(* Logix 5000 project; controller PBS_Perfusion vendor 1 type 14 code 217 rev 32.14; software revision 32.03; part 13 of 27 *)
(* tags used below, declared in another part *)
   Inp_PV : BOOL;   // Input Signal (process variable) from Sensor
   Inp_PVNotify : DINT;   // Related PV object alarm prio and ack status (enum)
   Inp_Target : BOOL;   // Target State of Input (Disagree Status if not in Target State)
   Cfg_NoSubstPV : BOOL;   // 1=Disallow selection of Substitute PV
   Cfg_Debounce : REAL;   // Minimum time Input Sts must maintain state (sec)
   Set_SimPV : BOOL;   // PV used in Simulation (Inp_Sim=1)
   Sts : BOOL;   // Discrete Input Status (incl. Debounce, Manual Override, if used)
   Sts_PV : BOOL;   // Discrete Input Status (actual, not subject to Override)
   Sts_SubstPV : BOOL;   // 1=Using Substitute PV (Input being overridden)
   Sts_InpPV : BOOL;   // 1=Using Input PV (normal)
   Sts_PVBad : BOOL;   // Input Comm Status/ Quality (0=OK, 1=Bad)
   Sts_TgtDisagreeCmp : ALIAS FOR TgtDisagreeGate.Inp;   // Input vs. Target comparicon result 1=Disagree
   Sts_TgtDisagree : ALIAS FOR TgtDisagree.Inp;   // 1=Input is not in Target state
   P_DIn : BOOL;   // Unique Parameter Name for auto - discovery
   Wrk_Status : BOOL;   // Internal Status (after Manual Override selection)
   TgtDisagree : P_Alarm;   // Target Disagree Alarm
   Wrk_FallT : TIMER;   // Timer to ensure Status LOW time on falling edge
   Wrk_RiseT : TIMER;   // Timer to ensure Status HIGH time on rising edge
   Wrk_SubstPV : BOOL;   // Internal flag: Using Substitute PV
   Wrk_Sts : DINT;   // Buffer for building Val_Sts
   TgtDisagreeGate : P_Gate;   // Target Disagree Condition Gate/Delay
   MCmd_InpPV : BOOL;   // Maintenance Command to use Input PV (normal)
   MCmd_SubstPV : BOOL;   // Maintenance Command to use Substitute PV (override input)
   MRdy_InpPV : BOOL;   // 1=Ready for MCmd_InpPV (enables HMI button)
   MRdy_SubstPV : BOOL;   // 1=Ready for MCmd_SubstPV (enables HMI button)
   MSet_SubstPV : BOOL;   // Maintenance-Entered Substitute PV
   Wrk_ErrDebounce : BOOL;   // Error in Debounce Timer configuration
   REAL : DINT;
(* P_DIn, continued *)

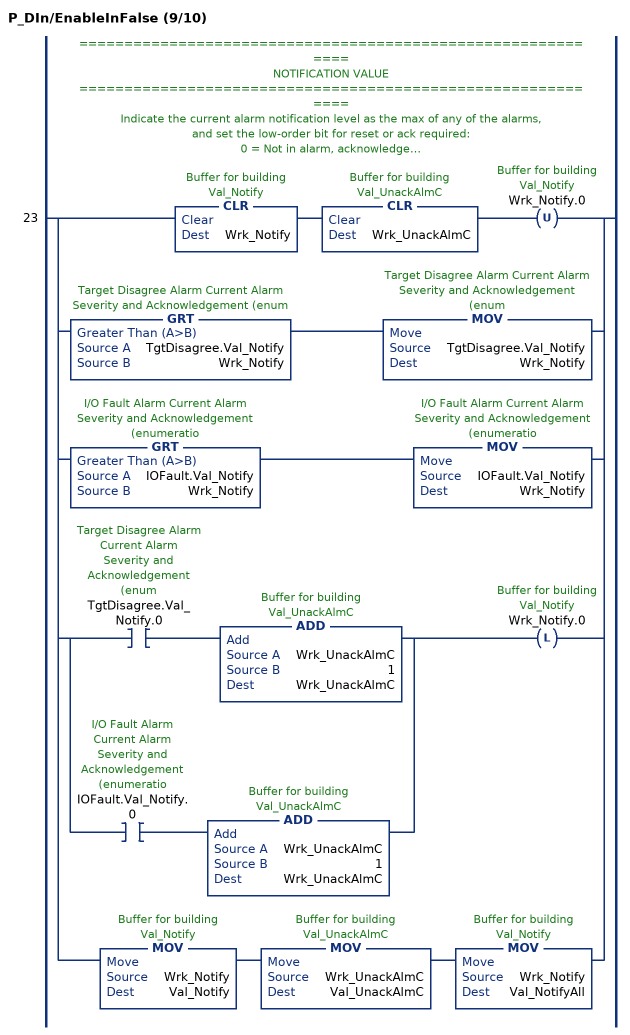
   // ============================================================
   // NOTIFICATION VALUE
   // ============================================================
   // Indicate the current alarm notification level as the max of any of the alarms,
   // and set the low-order bit for reset or ack required:
   // 0 = Not in alarm, acknowledged
   // 1 = Not in alarm, unacknowledged or reset required
   // 2 = Low severity alarm, acknowledged
   // 3 = Low severity alarm, unacknowledged
   // 4 = Medium severity alarm, acknowledged
   // 5 = Medium severity alarm, unacknowledged
   // 6 = High severity alarm, acknowledged
   // 7 = High severity alarm, unacknowledged
   // 8 = Urgent severity alarm, acknowledged
   // 9 = Urgent severity alarm, unacknowledged
   // #####  V4.00.00  2018-06-25:  Added Val_NotifyAll and Val_UnackAlmC to roll up alarm  #####
   // #####  priority / ack status and unack. alarm count.  #####
   // #####  Added I/O Fault alarm.  #####
   23: [CLR(Wrk_Notify) CLR(Wrk_UnackAlmC) OTU(Wrk_Notify.0) ,GRT(TgtDisagree.Val_Notify,Wrk_Notify) MOV(TgtDisagree.Val_Notify,Wrk_Notify) ,GRT(IOFault.Val_Notify,Wrk_Notify) MOV(IOFault.Val_Notify,Wrk_Notify) ,[XIC(TgtDisagree.Val_Notify.0) ADD(Wrk_UnackAlmC,1,Wrk_UnackAlmC) ,XIC(IOFault.Val_Notify.0) ADD(Wrk_UnackAlmC,1,Wrk_UnackAlmC) ] OTL(Wrk_Notify.0) ,MOV(Wrk_Notify,Val_Notify) MOV(Wrk_UnackAlmC,Val_UnackAlmC) MOV(Wrk_Notify,Val_NotifyAll) ];
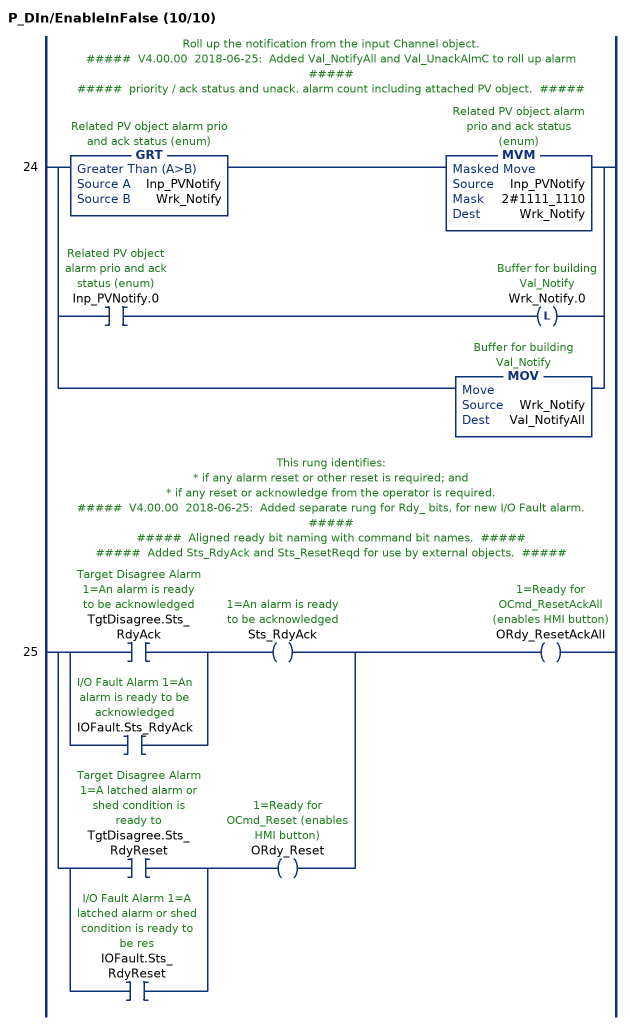
   // Roll up the notification from the input Channel object.
   // #####  V4.00.00  2018-06-25:  Added Val_NotifyAll and Val_UnackAlmC to roll up alarm  #####
   // #####  priority / ack status and unack. alarm count including attached PV object.  #####
   24: [GRT(Inp_PVNotify,Wrk_Notify) MVM(Inp_PVNotify,2#1111_1110,Wrk_Notify) ,XIC(Inp_PVNotify.0) OTL(Wrk_Notify.0) ,MOV(Wrk_Notify,Val_NotifyAll) ];
   // This rung identifies:
   // * if any alarm reset or other reset is required; and
   // * if any reset or acknowledge from the operator is required.
   // #####  V4.00.00  2018-06-25:  Added separate rung for Rdy_ bits, for new I/O Fault alarm.  #####
   // #####  Aligned ready bit naming with command bit names.  #####
   // #####  Added Sts_RdyAck and Sts_ResetReqd for use by external objects.  #####
   25: [[XIC(TgtDisagree.Sts_RdyAck) ,XIC(IOFault.Sts_RdyAck) ] OTE(Sts_RdyAck) ,[XIC(TgtDisagree.Sts_RdyReset) ,XIC(IOFault.Sts_RdyReset) ] OTE(ORdy_Reset) ]OTE(ORdy_ResetAckAll);
END_ROUTINE

ROUTINE Logic   (* ladder *)
// Normal Scan - status is updated and alarms are generated
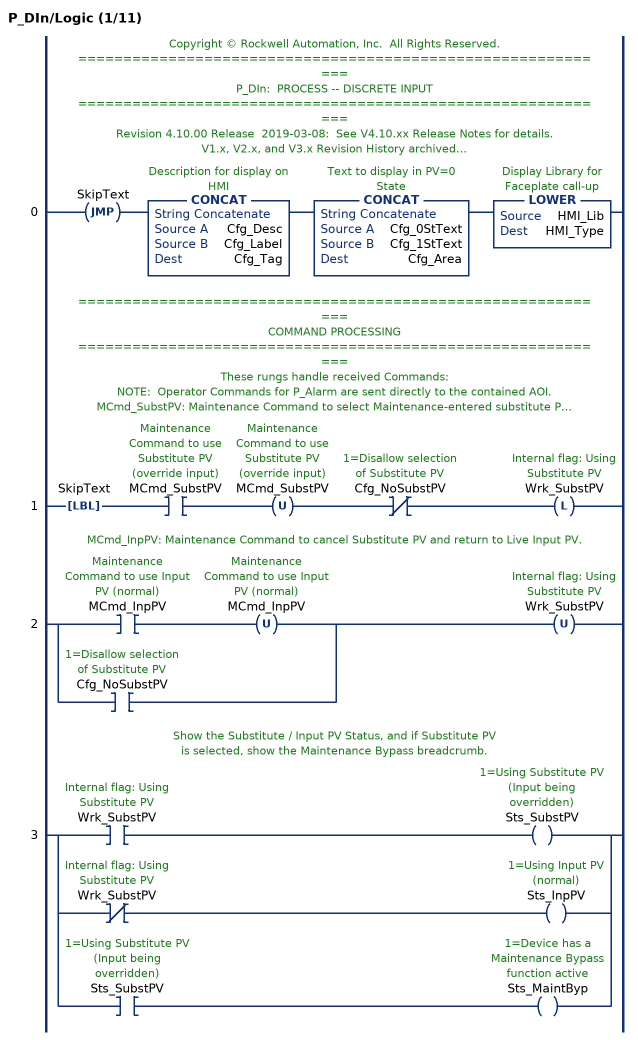
   // Copyright © Rockwell Automation, Inc.  All Rights Reserved.
   // ============================================================
   // P_DIn:  PROCESS -- DISCRETE INPUT
   // ============================================================
   // Revision 4.10.00 Release  2019-03-08:  See V4.10.xx Release Notes for details.
   // V1.x, V2.x, and V3.x Revision History archived.
   // V4.00.00  2018-06-25:  Added I/O Fault alarm.
   // Changed Inf_ items to HMI_, and added Cfg_Area for security.
   // Added notify and unack count rollup for Channel object.
   // Deleted Cfg_PCmdClear.  All Program Commands are now self-clearing.
   // Aligned ready bit naming with command bit names.
   // All OCmds/MCmds and ORdys/MRdys are now Local Tags.
   // Added Sts_RdyAck and Sts_ResetReqd for use by external objects.
   // Changed delay time configuration items to REAL seconds.
   // V4.10.00  2019-03-08:  Added Cfg_HasMoreObj.
   // ============================================================
   // This Instruction monitors a Discrete Input from a flow switch, motor vibration
   // switch, or any other discrete signal, and provides:
   // *  PV Status, with configurable names for the 0- and 1-states
   // * Input debounce for both the rising and falling transitions of the PV input
   // * An I/O Fault input.  An I/O Fault Alarm is raised when this input is true
   // *  A "Target" input -- the Target Disagree Alarm is raised when the PV input is not in
   // the same state as the Target for a configurable period of time
   // *  A Target Disagree "Gate" signal (with delay), used to enable the Alarm under
   // appropriate process conditions
   // * Commands to inhibit or enable alarms
   // * Setting of a simulated input signal for process simulation
   // * Selection of Substitute PV (by Maintenance personnel) or normal PV
   // Alarms are provided by P_Alarm AOI instances.
   // Target Disagree Status gating is provided by a P_Gate AOI instance.
   // ============================================================
   // SHOW LOCAL STRINGS
   // ============================================================
   // The STRINGs containing the text associated with each instance of this
   // instruction cannot be Input or Output Parameters, because STRINGs are not
   //  'atomic' types. (Inputs and Outputs must be SINT, INT, DINT, REAL, or BOOL.)
   // In order to make it easier to find and configure these STRINGs, this rung
   // was added.  THE JMP (and the LBL on the following rung)
   // MUST NOT BE REMOVED!!!
   // To view the STRINGs, go to the instruction instance (in LD or FBD), RIGHT-click
   // to bring up the context menu and select "Open Instruction Logic".
   // This rung will appear with the STRING values for the selected instance.
   // You may double-click the STRING values here to modify them as well.
   // #####  V4.00.00  2018-06-25:  Added string for Cfg_Area, renamed Inf_* to HMI_*.  #####
   0: JMP(SkipText)CONCAT(Cfg_Desc,Cfg_Label,Cfg_Tag)CONCAT(Cfg_0StText,Cfg_1StText,Cfg_Area)LOWER(HMI_Lib,HMI_Type);
   // ============================================================
   // COMMAND PROCESSING
   // ============================================================
   // These rungs handle received Commands:
   // NOTE:  Operator Commands for P_Alarm are sent directly to the contained AOI.
   // MCmd_SubstPV: Maintenance Command to select Maintenance-entered substitute PV
   // Do not allow this Command if Cfg_NoSubstPV is set.
   1: LBL(SkipText)XIC(MCmd_SubstPV)OTU(MCmd_SubstPV)XIO(Cfg_NoSubstPV)OTL(Wrk_SubstPV);
   // MCmd_InpPV: Maintenance Command to cancel Substitute PV and return to Live Input PV.
   2: [XIC(MCmd_InpPV) OTU(MCmd_InpPV) ,XIC(Cfg_NoSubstPV) ]OTU(Wrk_SubstPV);
   // Show the Substitute / Input PV Status, and if Substitute PV
   // is selected, show the Maintenance Bypass breadcrumb.
   3: [XIC(Wrk_SubstPV) OTE(Sts_SubstPV) ,XIO(Wrk_SubstPV) OTE(Sts_InpPV) ,XIC(Sts_SubstPV) OTE(Sts_MaintByp) ];
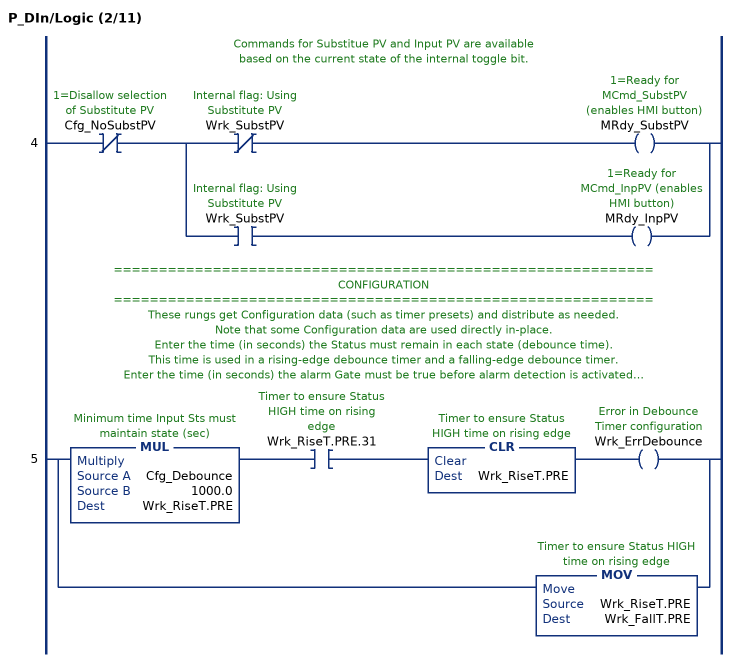
   // Commands for Substitue PV and Input PV are available
   // based on the current state of the internal toggle bit.
   4: XIO(Cfg_NoSubstPV)[XIO(Wrk_SubstPV) OTE(MRdy_SubstPV) ,XIC(Wrk_SubstPV) OTE(MRdy_InpPV) ];
   // ============================================================
   // CONFIGURATION
   // ============================================================
   // These rungs get Configuration data (such as timer presets) and distribute as needed.
   // Note that some Configuration data are used directly in-place.
   // Enter the time (in seconds) the Status must remain in each state (debounce time).
   // This time is used in a rising-edge debounce timer and a falling-edge debounce timer.
   // Enter the time (in seconds) the alarm Gate must be true before alarm detection is activated.
   // Enter the On-Delay and Off-Delay times (in seconds) for the Target Disagree Status
   // (which feeds the Target Disagree Alarm).
   // If the timer preset calcuated wraps negative (more than 2.14... million seconds), then establish
   // a valid limit value for the Preset.  Note that a negative timer preset will fault the controller!!!
   // #####  V4.00.00  2018-06-25:  Changed delay time configuration items to REAL seconds.  #####
   5: [MUL(Cfg_Debounce,1000.0,Wrk_RiseT.PRE) XIC(Wrk_RiseT.PRE.31) CLR(Wrk_RiseT.PRE) OTE(Wrk_ErrDebounce) ,MOV(Wrk_RiseT.PRE,Wrk_FallT.PRE) ];
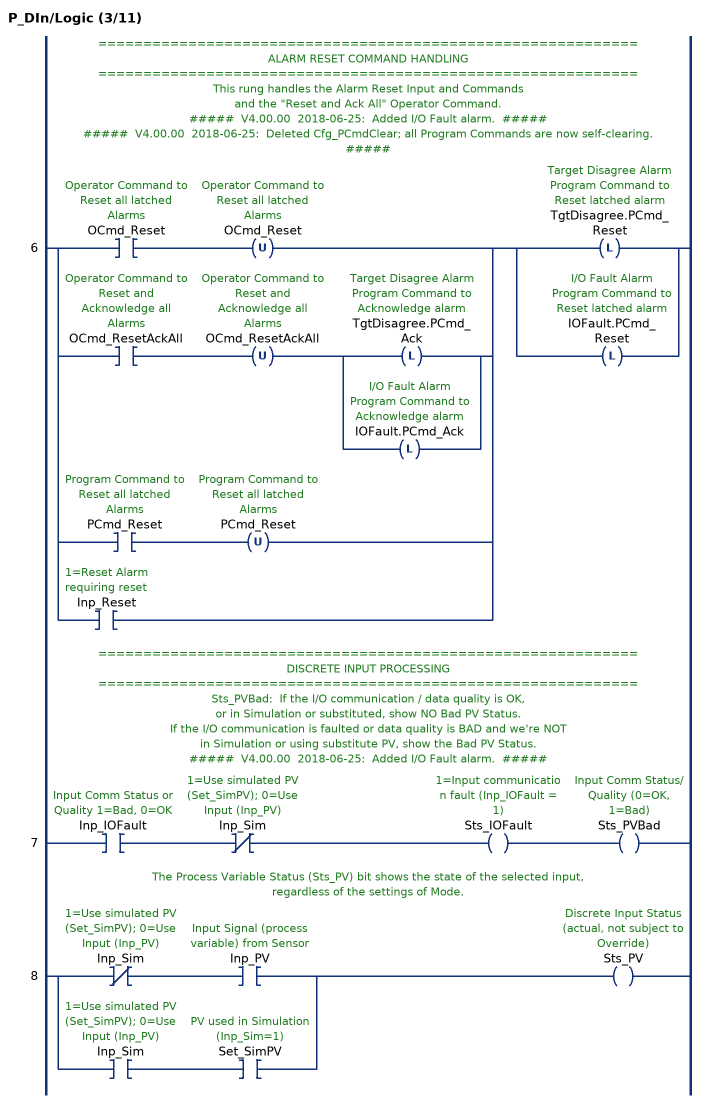
   // ============================================================
   // ALARM RESET COMMAND HANDLING
   // ============================================================
   // This rung handles the Alarm Reset Input and Commands
   // and the "Reset and Ack All" Operator Command.
   // #####  V4.00.00  2018-06-25:  Added I/O Fault alarm.  #####
   // #####  V4.00.00  2018-06-25:  Deleted Cfg_PCmdClear; all Program Commands are now self-clearing.  #####
   6: [XIC(OCmd_Reset) OTU(OCmd_Reset) ,XIC(OCmd_ResetAckAll) OTU(OCmd_ResetAckAll) [OTL(TgtDisagree.PCmd_Ack) ,OTL(IOFault.PCmd_Ack) ] ,XIC(PCmd_Reset) OTU(PCmd_Reset) ,XIC(Inp_Reset) ][OTL(TgtDisagree.PCmd_Reset) ,OTL(IOFault.PCmd_Reset) ];
   // ============================================================
   // DISCRETE INPUT PROCESSING
   // ============================================================
   // Sts_PVBad:  If the I/O communication / data quality is OK,
   // or in Simulation or substituted, show NO Bad PV Status.
   // If the I/O communication is faulted or data quality is BAD and we're NOT
   // in Simulation or using substitute PV, show the Bad PV Status.
   // #####  V4.00.00  2018-06-25:  Added I/O Fault alarm.  #####
   7: XIC(Inp_IOFault)XIO(Inp_Sim)OTE(Sts_IOFault)OTE(Sts_PVBad);
   // The Process Variable Status (Sts_PV) bit shows the state of the selected input,
   // regardless of the settings of Mode.
   8: [XIO(Inp_Sim) XIC(Inp_PV) ,XIC(Inp_Sim) XIC(Set_SimPV) ]OTE(Sts_PV);
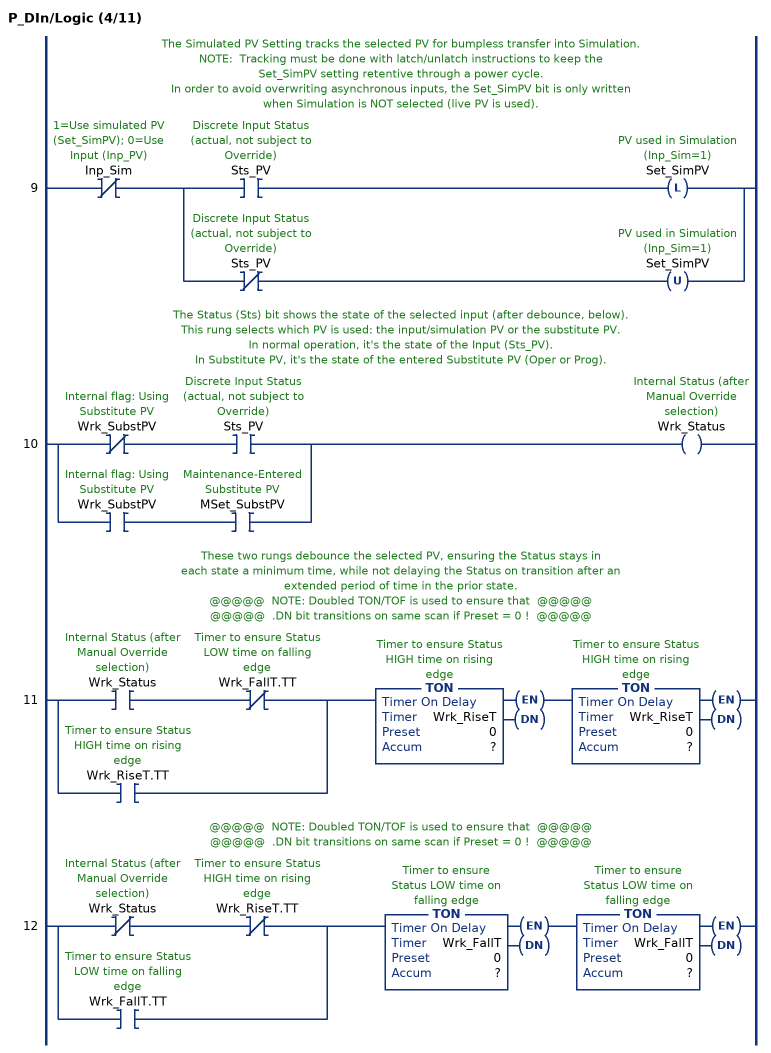
   // The Simulated PV Setting tracks the selected PV for bumpless transfer into Simulation.
   // NOTE:  Tracking must be done with latch/unlatch instructions to keep the
   // Set_SimPV setting retentive through a power cycle.
   // In order to avoid overwriting asynchronous inputs, the Set_SimPV bit is only written
   // when Simulation is NOT selected (live PV is used).
   9: XIO(Inp_Sim)[XIC(Sts_PV) OTL(Set_SimPV) ,XIO(Sts_PV) OTU(Set_SimPV) ];
   // The Status (Sts) bit shows the state of the selected input (after debounce, below).
   // This rung selects which PV is used: the input/simulation PV or the substitute PV.
   // In normal operation, it's the state of the Input (Sts_PV).
   // In Substitute PV, it's the state of the entered Substitute PV (Oper or Prog).
   10: [XIO(Wrk_SubstPV) XIC(Sts_PV) ,XIC(Wrk_SubstPV) XIC(MSet_SubstPV) ]OTE(Wrk_Status);
   // These two rungs debounce the selected PV, ensuring the Status stays in
   // each state a minimum time, while not delaying the Status on transition after an
   // extended period of time in the prior state.
   // @@@@@  NOTE: Doubled TON/TOF is used to ensure that  @@@@@
   // @@@@@  .DN bit transitions on same scan if Preset = 0 !  @@@@@
   11: [XIC(Wrk_Status) XIO(Wrk_FallT.TT) ,XIC(Wrk_RiseT.TT) ]TON(Wrk_RiseT,?,?)TON(Wrk_RiseT,?,?);
   // @@@@@  NOTE: Doubled TON/TOF is used to ensure that  @@@@@
   // @@@@@  .DN bit transitions on same scan if Preset = 0 !  @@@@@
   12: [XIO(Wrk_Status) XIO(Wrk_RiseT.TT) ,XIC(Wrk_FallT.TT) ]TON(Wrk_FallT,?,?)TON(Wrk_FallT,?,?);
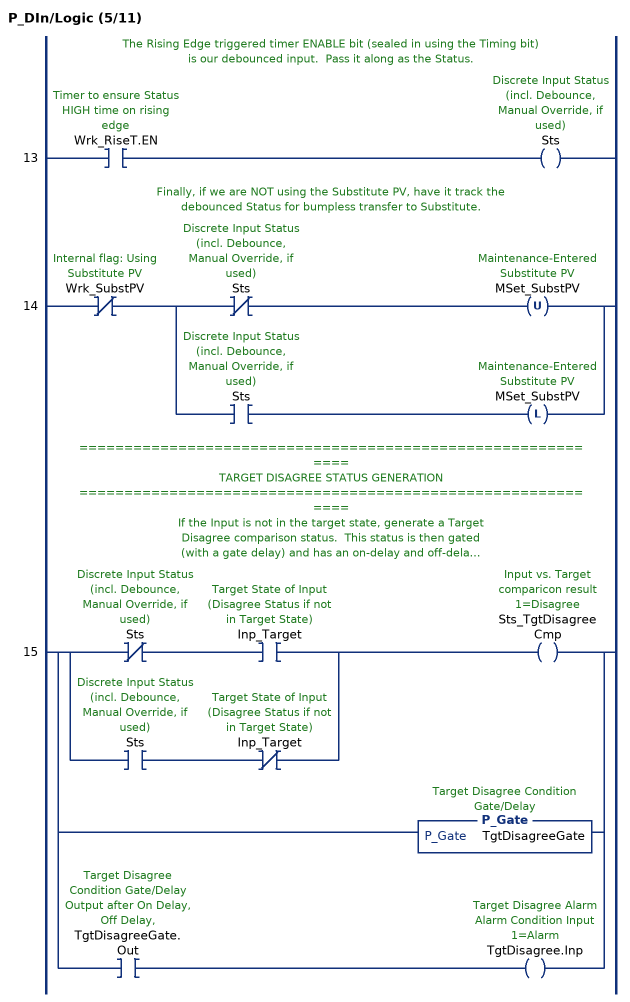
   // The Rising Edge triggered timer ENABLE bit (sealed in using the Timing bit)
   // is our debounced input.  Pass it along as the Status.
   13: XIC(Wrk_RiseT.EN)OTE(Sts);
   // Finally, if we are NOT using the Substitute PV, have it track the
   // debounced Status for bumpless transfer to Substitute.
   14: XIO(Wrk_SubstPV)[XIO(Sts) OTU(MSet_SubstPV) ,XIC(Sts) OTL(MSet_SubstPV) ];
   // ============================================================
   // TARGET DISAGREE STATUS GENERATION
   // ============================================================
   // If the Input is not in the target state, generate a Target
   // Disagree comparison status.  This status is then gated
   // (with a gate delay) and has an on-delay and off-delay
   // before feeding the final Target Disagree status bit.
   15: [[XIO(Sts) XIC(Inp_Target) ,XIC(Sts) XIO(Inp_Target) ] OTE(Sts_TgtDisagreeCmp) ,P_Gate(TgtDisagreeGate) ,XIC(TgtDisagreeGate.Out) OTE(TgtDisagree.Inp) ];
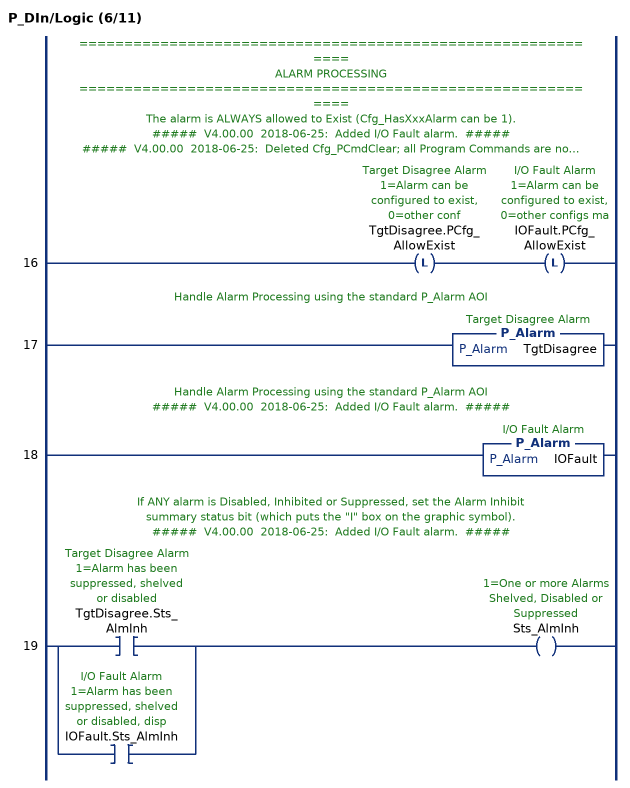
   // ============================================================
   // ALARM PROCESSING
   // ============================================================
   // The alarm is ALWAYS allowed to Exist (Cfg_HasXxxAlarm can be 1).
   // #####  V4.00.00  2018-06-25:  Added I/O Fault alarm.  #####
   // #####  V4.00.00  2018-06-25:  Deleted Cfg_PCmdClear; all Program Commands are now self-clearing.  #####
   16: OTL(TgtDisagree.PCfg_AllowExist)OTL(IOFault.PCfg_AllowExist);
   // Handle Alarm Processing using the standard P_Alarm AOI
   17: P_Alarm(TgtDisagree);
   // Handle Alarm Processing using the standard P_Alarm AOI
   // #####  V4.00.00  2018-06-25:  Added I/O Fault alarm.  #####
   18: P_Alarm(IOFault);
   // If ANY alarm is Disabled, Inhibited or Suppressed, set the Alarm Inhibit
   // summary status bit (which puts the "I" box on the graphic symbol).
   // #####  V4.00.00  2018-06-25:  Added I/O Fault alarm.  #####
   19: [XIC(TgtDisagree.Sts_AlmInh) ,XIC(IOFault.Sts_AlmInh) ]OTE(Sts_AlmInh);
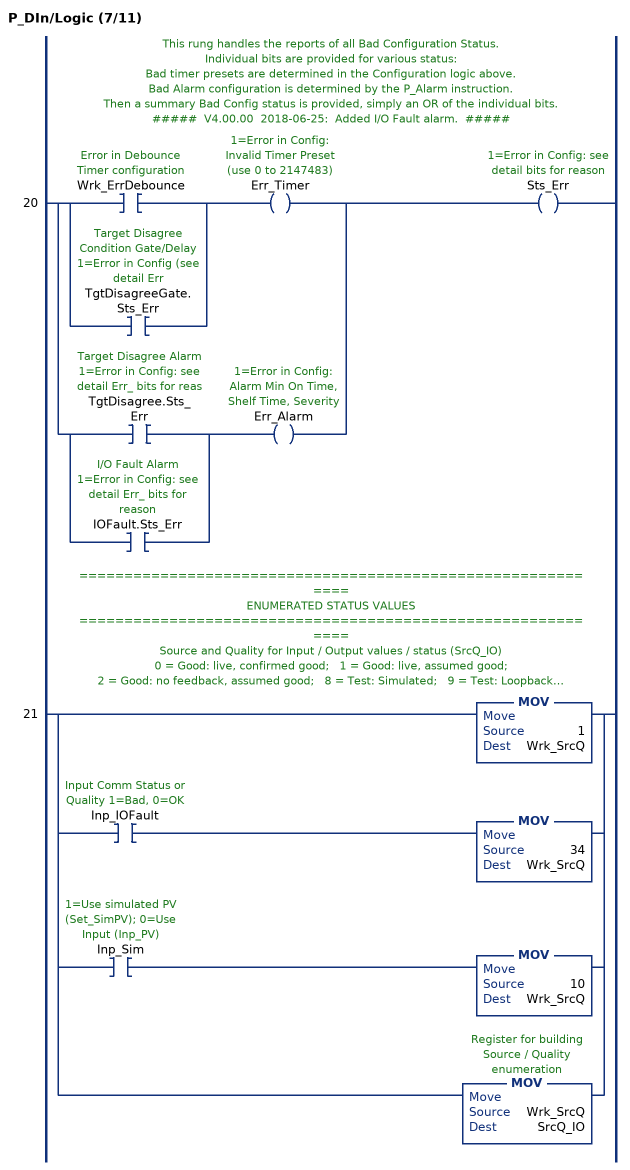
   // This rung handles the reports of all Bad Configuration Status.
   // Individual bits are provided for various status:
   // Bad timer presets are determined in the Configuration logic above.
   // Bad Alarm configuration is determined by the P_Alarm instruction.
   // Then a summary Bad Config status is provided, simply an OR of the individual bits.
   // #####  V4.00.00  2018-06-25:  Added I/O Fault alarm.  #####
   20: [[XIC(Wrk_ErrDebounce) ,XIC(TgtDisagreeGate.Sts_Err) ] OTE(Err_Timer) ,[XIC(TgtDisagree.Sts_Err) ,XIC(IOFault.Sts_Err) ] OTE(Err_Alarm) ]OTE(Sts_Err);
   // ============================================================
   // ENUMERATED STATUS VALUES
   // ============================================================
   // Source and Quality for Input / Output values / status (SrcQ_IO)
   // 0 = Good: live, confirmed good;   1 = Good: live, assumed good;
   // 2 = Good: no feedback, assumed good;   8 = Test: Simulated;   9 = Test: Loopback;
   // 10 = Test: Manually Entered;   16 = Uncertain: Live, off-spec;
   // 17 = Uncertain, Substituted at Device / Bus;   18 = Uncertain, Substituted at AOI;
   // 19 = Uncertain, using last known good;    20 = Uncertain, using replacement value;
   // 32 = Bad, Signal Failure;   33 = Bad, Channel Fault;
   // 34 = Bad, Module / Comms Fault;   35 = Bad, Invalid Configuration
   // #####  V4.00.00  2018-06-25:  Added I/O Fault alarm.  #####
   21: [MOV(1,Wrk_SrcQ) ,XIC(Inp_IOFault) MOV(34,Wrk_SrcQ) ,XIC(Inp_Sim) MOV(10,Wrk_SrcQ) ,MOV(Wrk_SrcQ,SrcQ_IO) ];
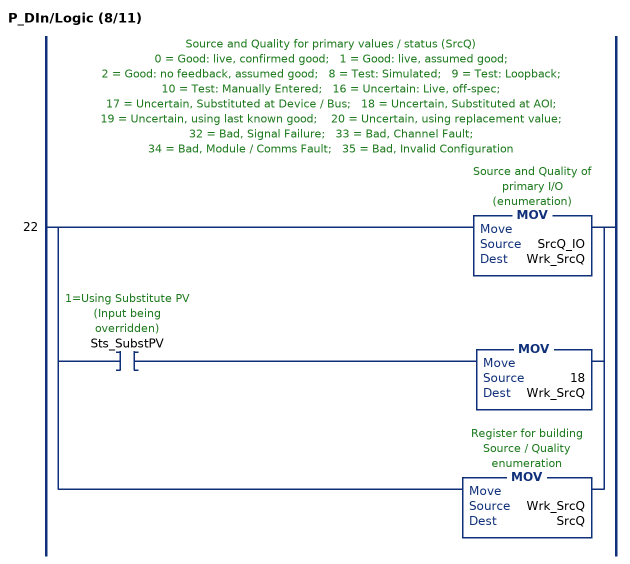
   // Source and Quality for primary values / status (SrcQ)
   // 0 = Good: live, confirmed good;   1 = Good: live, assumed good;
   // 2 = Good: no feedback, assumed good;   8 = Test: Simulated;   9 = Test: Loopback;
   // 10 = Test: Manually Entered;   16 = Uncertain: Live, off-spec;
   // 17 = Uncertain, Substituted at Device / Bus;   18 = Uncertain, Substituted at AOI;
   // 19 = Uncertain, using last known good;    20 = Uncertain, using replacement value;
   // 32 = Bad, Signal Failure;   33 = Bad, Channel Fault;
   // 34 = Bad, Module / Comms Fault;   35 = Bad, Invalid Configuration
   22: [MOV(SrcQ_IO,Wrk_SrcQ) ,XIC(Sts_SubstPV) MOV(18,Wrk_SrcQ) ,MOV(Wrk_SrcQ,SrcQ) ];
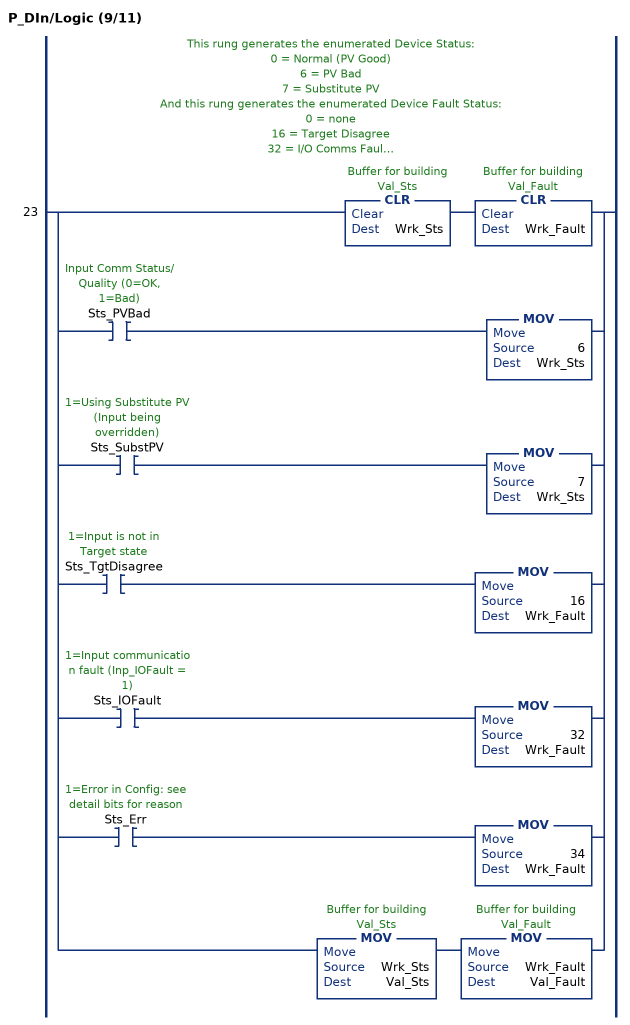
   // This rung generates the enumerated Device Status:
   // 0 = Normal (PV Good)
   // 6 = PV Bad
   // 7 = Substitute PV
   // And this rung generates the enumerated Device Fault Status:
   // 0 = none
   // 16 = Target Disagree
   // 32 = I/O Comms Fault
   // 34 = Config Error
   // #####  V4.00.00  2018-06-25:  Added I/O Fault alarm.  #####
   23: [CLR(Wrk_Sts) CLR(Wrk_Fault) ,XIC(Sts_PVBad) MOV(6,Wrk_Sts) ,XIC(Sts_SubstPV) MOV(7,Wrk_Sts) ,XIC(Sts_TgtDisagree) MOV(16,Wrk_Fault) ,XIC(Sts_IOFault) MOV(32,Wrk_Fault) ,XIC(Sts_Err) MOV(34,Wrk_Fault) ,MOV(Wrk_Sts,Val_Sts) MOV(Wrk_Fault,Val_Fault) ];
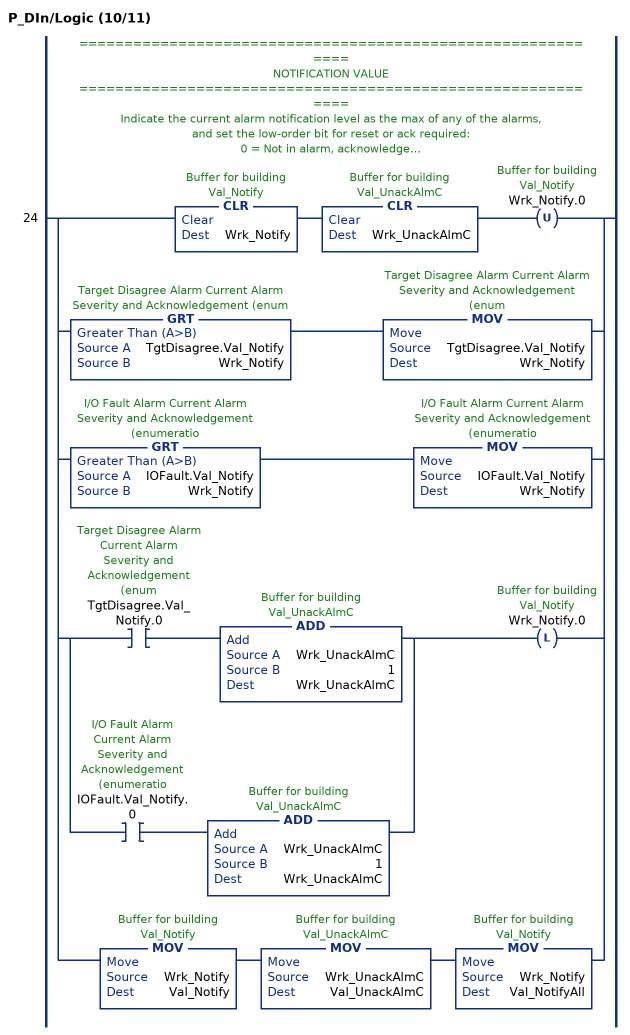
   // ============================================================
   // NOTIFICATION VALUE
   // ============================================================
   // Indicate the current alarm notification level as the max of any of the alarms,
   // and set the low-order bit for reset or ack required:
   // 0 = Not in alarm, acknowledged
   // 1 = Not in alarm, unacknowledged or reset required
   // 2 = Low severity alarm, acknowledged
   // 3 = Low severity alarm, unacknowledged
   // 4 = Medium severity alarm, acknowledged
   // 5 = Medium severity alarm, unacknowledged
   // 6 = High severity alarm, acknowledged
   // 7 = High severity alarm, unacknowledged
   // 8 = Urgent severity alarm, acknowledged
   // 9 = Urgent severity alarm, unacknowledged
   // #####  V4.00.00  2018-06-25:  Added Val_NotifyAll and Val_UnackAlmC to roll up alarm  #####
   // #####  priority / ack status and unack. alarm count.  #####
   // #####  Added I/O Fault alarm.  #####
   24: [CLR(Wrk_Notify) CLR(Wrk_UnackAlmC) OTU(Wrk_Notify.0) ,GRT(TgtDisagree.Val_Notify,Wrk_Notify) MOV(TgtDisagree.Val_Notify,Wrk_Notify) ,GRT(IOFault.Val_Notify,Wrk_Notify) MOV(IOFault.Val_Notify,Wrk_Notify) ,[XIC(TgtDisagree.Val_Notify.0) ADD(Wrk_UnackAlmC,1,Wrk_UnackAlmC) ,XIC(IOFault.Val_Notify.0) ADD(Wrk_UnackAlmC,1,Wrk_UnackAlmC) ] OTL(Wrk_Notify.0) ,MOV(Wrk_Notify,Val_Notify) MOV(Wrk_UnackAlmC,Val_UnackAlmC) MOV(Wrk_Notify,Val_NotifyAll) ];
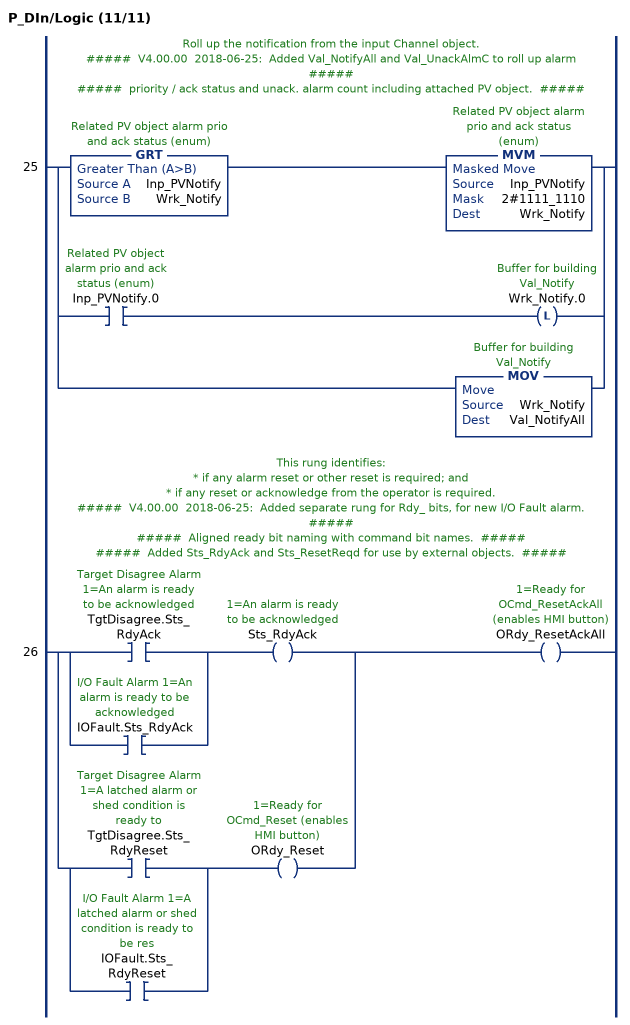
   // Roll up the notification from the input Channel object.
   // #####  V4.00.00  2018-06-25:  Added Val_NotifyAll and Val_UnackAlmC to roll up alarm  #####
   // #####  priority / ack status and unack. alarm count including attached PV object.  #####
   25: [GRT(Inp_PVNotify,Wrk_Notify) MVM(Inp_PVNotify,2#1111_1110,Wrk_Notify) ,XIC(Inp_PVNotify.0) OTL(Wrk_Notify.0) ,MOV(Wrk_Notify,Val_NotifyAll) ];
   // This rung identifies:
   // * if any alarm reset or other reset is required; and
   // * if any reset or acknowledge from the operator is required.
   // #####  V4.00.00  2018-06-25:  Added separate rung for Rdy_ bits, for new I/O Fault alarm.  #####
   // #####  Aligned ready bit naming with command bit names.  #####
   // #####  Added Sts_RdyAck and Sts_ResetReqd for use by external objects.  #####
   26: [[XIC(TgtDisagree.Sts_RdyAck) ,XIC(IOFault.Sts_RdyAck) ] OTE(Sts_RdyAck) ,[XIC(TgtDisagree.Sts_RdyReset) ,XIC(IOFault.Sts_RdyReset) ] OTE(ORdy_Reset) ]OTE(ORdy_ResetAckAll);
END_ROUTINE

ROUTINE Prescan   (* ladder *)
// Clear "lurking" Commands
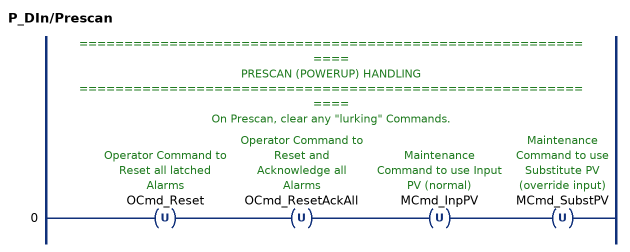
   // ============================================================
   // PRESCAN (POWERUP) HANDLING
   // ============================================================
   // On Prescan, clear any "lurking" Commands.
   0: OTU(OCmd_Reset)OTU(OCmd_ResetAckAll)OTU(MCmd_InpPV)OTU(MCmd_SubstPV);
END_ROUTINE
END_ADD_ON_INSTRUCTION

ADD_ON_INSTRUCTION P_DOut   (* revision 4.10 .01 Release, vendor Rockwell Automation, ExecutePrescan, ExecuteEnableInFalse *)
// Discrete Output
// Revision note:
// See Instruction Help for a summary of changes, and see 4.10 Release Notes for details.
// Help:
// Copyright © Rockwell Automation, Inc.  All Rights Reserved.
// This Instruction controls (and optionally monitors feedback for)
// a single Discrete Output and provides:
// *  Operator and Program Commands to:
//     -  turn the output ON
//     -  turn the output OFF
//     -  if the output is OFF, pulse it ON for a configured time
//     -  if the output is ON, pulse it OFF for a configured time, and
//     -  pulse the output continuously at the configured ON
//         and OFF times (e.g., for blinking a lamp)
// *  User-configurable ON delay and OFF delay before first output change
// *  User-configurable text labels for the ON and OFF states
// *  Optional monitoring of ON and OFF state confirmation feedbacks
// *  Detection of Failure to turn ON or OFF (when feedbacks are used)
// *  Monitoring of Permissive conditions to allow energizing output
// *  Monitoring of Interlock conditions to de-energize output
// *  Simulation, providing feedback of a working device while
//       disabling output (keeping de-energized)
// *  Monitoring of I/O communication faults
// *  Alarms for Fail to Turn ON, Fail to turn OFF (if feedbacks are
//       used), Interlock Trip, I/O Fault
// *  "NotReady" status for display on Graphic Symbol and "Available"
//      status for use by automation logic to know whether output can be
//      controlled by other objects.
// Command Sources are arbitrated by a P_CmdSrc Add-On Instruction instance.
// Command Sources: Operator, Program, External, Override, Maintenance, Out of
// Service, Hand.  Alarms are provided by P_Alarm Add-On Instruction instances.
// SUMMARY OF CHANGES FROM PREVIOUS VERSION (4.10.00)
// * Corrected operation of state machine with alert horn.
// SUMMARY OF CHANGES FROM PREVIOUS VERSION (4.00.02)
// See 4.10 Release Notes for details.
// * Added audible alert on commanded energize/state change.
// * Added Horn Status, Horn Inhibit.
// * Changed availability to use input availability from interlocks.
// * Updated to P_CmdSrc V4.10.00.
// * Added Cfg_HasMoreObj.
// SUMMARY OF CHANGES FROM PREVIOUS VERSION (4.00.00)
// See 4.00 Release Notes for details.
// * Fixed feedback determination for simulation or no feedback.
// SUMMARY OF CHANGES FROM PREVIOUS VERSION (3.5-11)
// See 4.00 Release Notes for details.
// * Changed Inf_ items to HMI_, and added Cfg_Area for security.
// * Added notify and unack count rollup for associated object(s).
// * Changed "Mode" to "Command Source" using P_CmdSrc 4.00.00.
// * Deleted Cfg_PCmdClear; all Program Commands are now self-clearing.
// * Added option Cfg_HasPulse to enable or disable pulsing functions.
// * Aligned ready bit naming with command bit names.
// * All OCmds/MCmds and ORdys/MRdys are now Local Tags.
// * Added Sts_RdyAck and Sts_RdyReset for use by external objects.
// * Changed delay / time configuration items to REAL seconds.
VAR_INPUT
   Inp_OnFdbk : BOOL; {visible}   // Input Signal: ON feedback from device
   Inp_OffFdbk : BOOL; {visible}   // Input Signal: OFF feedback from device
   Inp_PermOK : BOOL := 1; {visible}   // 1=ON Permissives OK, device can turn ON
   Inp_NBPermOK : BOOL := 1; {visible}   // 1=Non-Bypassable ON Permissives OK, device can turn ON
   Inp_IntlkOK : BOOL := 1; {visible}   // 1=Interlocks OK, device can turn ON and stay ON
   Inp_NBIntlkOK : BOOL := 1; {visible}   // 1=Non-Bypassable Interlocks OK, device can turn ON and stay ON
   Inp_IntlkAvail : BOOL;   // 1 = Interlock Availibility OK
   Inp_IOFault : BOOL;   // Input Communication Status 0=OK, 1=fail
   Inp_Sim : BOOL;   // 1=Simulate working device; 0=Turn ON/OFF actual device
   Inp_Hand : ALIAS FOR CmdSrc.Inp_Hand;
   Inp_Ovrd : ALIAS FOR CmdSrc.Inp_Ovrd;
   Inp_OvrdCmd : DINT;   // Ovrd Device Command 0=None, 1=Off, 2=On, 3=Pulse Off, 4=Pulse On, 5=Pulse Cont
   Inp_ExtInh : ALIAS FOR CmdSrc.Inp_ExtInh;
   Inp_HornInh : BOOL;   // 1 = Inhibit audible alert, 0 = Alllow audible alert
   Inp_Reset : BOOL;   // 1=Reset Shed Latches and Cleared Alarms
   Cfg_HasPulse : BOOL;   // 1=Enable pulsing functions, 0=On/Off only
   Cfg_CompletePulse : BOOL;   // 1=Finish Pulse when commanded ON or OFF; 0=switch immediately
   Cfg_HasOnFdbk : BOOL;   // 1=Device provides an ON feedback signal
   Cfg_HasOffFdbk : BOOL;   // 1=Device provides an OFF feedback signal
   Cfg_UseOnFdbk : BOOL;   // 1=Device ON feedback should be used for failure checking
   Cfg_UseOffFdbk : BOOL;   // 1=Device OFF feedback should be used for failure checking
   Cfg_FdbkFail : BOOL;   // 1=Both feedbacks ON is invalid; 0=Both feedbacks OFF is invalid
   Cfg_HasPermObj : BOOL;   // 1=Tells HMI a P_Perm is connected to Inp_Perm
   Cfg_HasIntlkObj : BOOL;   // 1=Tells HMI a P_Intlk is connected to Inp_Intlk
   Cfg_HasMoreObj : BOOL;   // 1=Tells HMI an object with more info is available
   Cfg_HornOnChange : BOOL;   // 0 = Horn on energize only, 1 = Horn on any state change
   Cfg_OperOffPrio : BOOL;   // 1=OCmd_Off any time, 0=OCmd_Off only when Oper selected
   Cfg_ExtOffPrio : BOOL;   // 1=XCmd_Off any time, 0=XCmd_Off only when Oper selected
   Cfg_OCmdResets : BOOL;   // 1=New device OCmd resets shed latches and cleared alarms, 0=OCmdReset req'd.
   Cfg_XCmdResets : BOOL;   // 1=New device XCmd resets shed latches and cleared alarms, 0=XCmdReset req'd.
   Cfg_OvrdPermIntlk : BOOL;   // 1=Override ignores Bypassable Perm/ Intlk; 0=always use Perm/Intlk
   Cfg_ShedOnFail : BOOL := 1;   // 1=Go to State 0 and Alarm on Fail to reach position; 0=Alarm only on Fail
   Cfg_ShedOnIOFault : BOOL := 1;   // 1=Go to State 0 and Alarm on I/O Fault; 0=Alarm only on I/O Fault
   Cfg_HasOnFailAlm : ALIAS FOR OnFail.Cfg_Exists;   // 1=Fail to Turn ON Alarm exists and will be checked
   Cfg_HasOffFailAlm : ALIAS FOR OffFail.Cfg_Exists;   // 1=Fail to Turn OFF Alarm exists and will be checked
   Cfg_HasIntlkTripAlm : ALIAS FOR IntlkTrip.Cfg_Exists;   // 1=Interlock Trip Alarm exists and will be checked
   Cfg_HasIOFaultAlm : ALIAS FOR IOFault.Cfg_Exists;   // 1=I/O Fault Alarm exists and will be checked
   Cfg_OnFailResetReqd : ALIAS FOR OnFail.Cfg_ResetReqd;   // 1=Reset required to clear Fail to Turn ON Alarm
   Cfg_OffFailResetReqd : ALIAS FOR OffFail.Cfg_ResetReqd;   // 1=Reset required to clear Fail to Turn OFF Alarm
   Cfg_IntlkTripResetReqd : ALIAS FOR IntlkTrip.Cfg_ResetReqd;   // 1=Reset required to clear Interlock Trip Alarm
   Cfg_IOFaultResetReqd : ALIAS FOR IOFault.Cfg_ResetReqd;   // 1=Reset required to clear I/O Fault Alarm
   Cfg_OnFailAckReqd : ALIAS FOR OnFail.Cfg_AckReqd;   // 1=Acknowledge required for Fail to Turn ON Alarm
   Cfg_OffFailAckReqd : ALIAS FOR OffFail.Cfg_AckReqd;   // 1=Acknowledge required for Fail to Turn OFF Alarm
   Cfg_IntlkTripAckReqd : ALIAS FOR IntlkTrip.Cfg_AckReqd;   // 1=Acknowledge required for Interlock Trip Alarm
   Cfg_IOFaultAckReqd : ALIAS FOR IOFault.Cfg_AckReqd;   // 1=Acknowledge required for I/O Fault Alarm
   Cfg_OnFailSeverity : ALIAS FOR OnFail.Cfg_Severity;   // Fail To Turn OFF Alarm Severity: 1..250=Low, 251..500=Medium, 501..750=High, 751..1000=Urgent
   Cfg_OffFailSeverity : ALIAS FOR OffFail.Cfg_Severity;   // Fail To Turn ON Alarm Severity: 1..250=Low, 251..500=Medium, 501..750=High, 751..1000=Urgent
   Cfg_IntlkTripSeverity : ALIAS FOR IntlkTrip.Cfg_Severity;   // Interlock Trip Alarm Severity: 1..250=Low, 251..500=Medium, 501..750=High, 751..1000=Urgent
   Cfg_IOFaultSeverity : ALIAS FOR IOFault.Cfg_Severity;   // I/O Fault Alarm Severity: 1..250=Low, 251..500=Medium, 501..750=High, 751..1000=Urgent
   Cfg_StartHornT : REAL;   // Time to sound audible on commanded start (sec) (0=disabled)
   Cfg_SimFdbkT : REAL := 2.0;   // Delay to echo back of ON/OFF status when in Simulation (sec)
   Cfg_OnDelayT : REAL;   // Delay before initially turning output ON (sec)
   Cfg_OffDelayT : REAL;   // Delay before initially turning output OFF (sec)
   Cfg_OnPulseT : REAL := 0.5;   // Output ON time for Pulse ON or Pulse Continuous
   Cfg_OffPulseT : REAL := 0.5;   // Output OFF time for Pulse OFF or Pulse Continuous
   Cfg_OnFailT : REAL := 10.0;   // Time after Output ON to get ON Feedback before Fault (sec)
   Cfg_OffFailT : REAL := 10.0;   // Time after Output OFF to get OFF Feedback before Fault (sec)
   PSet_Owner : DINT;   // Program Owner Request ID (non-zero) or Release (zero)
   PCmd_On : BOOL;   // Program Command to turn device ON
   PCmd_Off : BOOL;   // Program Command to turn device OFF
   PCmd_OnPulse : BOOL;   // Program Command to pulse device (which is OFF) ON once
   PCmd_OffPulse : BOOL;   // Program Command to pulse device (which is ON) OFF once
   PCmd_ContPulse : BOOL;   // Program Command to pulse device continuously (blink)
   PCmd_Prog : ALIAS FOR CmdSrc.PCmd_Prog;
   PCmd_Oper : ALIAS FOR CmdSrc.PCmd_Oper;
   PCmd_Lock : ALIAS FOR CmdSrc.PCmd_Lock;
   PCmd_Unlock : ALIAS FOR CmdSrc.PCmd_Unlock;
   PCmd_Normal : ALIAS FOR CmdSrc.PCmd_Normal;
   PCmd_Reset : BOOL;   // Program Command to ResetShed Latches and Cleared Alarms
   PCmd_OnFailAck : ALIAS FOR OnFail.PCmd_Ack;   // Program Command to Acknowledge Fail to Turn ON Alarm
   PCmd_OnFailSuppress : ALIAS FOR OnFail.PCmd_Suppress;   // Program Command to Suppress Fail to Turn ON Alarm
   PCmd_OnFailUnsuppress : ALIAS FOR OnFail.PCmd_Unsuppress;   // Program Command to UnsuppressFail to Turn ON Alarm
   PCmd_OnFailUnshelve : ALIAS FOR OnFail.PCmd_Unshelve;   // Program Command to Unshelve Fail to Turn ON Alarm
   PCmd_OffFailAck : ALIAS FOR OffFail.PCmd_Ack;   // Program Command to Acknowledge Fail to Turn OFF Alarm
   PCmd_OffFailSuppress : ALIAS FOR OffFail.PCmd_Suppress;   // Program Command to Suppress Fail to Turn OFF Alarm
   PCmd_OffFailUnsuppress : ALIAS FOR OffFail.PCmd_Unsuppress;   // Program Command to Unsuppress Fail to Turn OFF Alarm
   PCmd_OffFailUnshelve : ALIAS FOR OffFail.PCmd_Unshelve;   // Program Command to Unshelve Failt to Turn OFF Alarm
   PCmd_IntlkTripAck : ALIAS FOR IntlkTrip.PCmd_Ack;   // Program Command to Acknowledge Interlock Trip Alarm
   PCmd_IntlkTripSuppress : ALIAS FOR IntlkTrip.PCmd_Suppress;   // Program Command to Suppress Interlock Trip Alarm
   PCmd_IntlkTripUnsuppress : ALIAS FOR IntlkTrip.PCmd_Unsuppress;   // Program Command to Unsuppress Interlock Trip Alarm
   PCmd_IntlkTripUnshelve : ALIAS FOR IntlkTrip.PCmd_Unshelve;   // Program Command to Unshelve Interlock Trip Alarm
   PCmd_IOFaultAck : ALIAS FOR IOFault.PCmd_Ack;   // Program Command to Acknowledge I/O Fault Alarm
   PCmd_IOFaultSuppress : ALIAS FOR IOFault.PCmd_Suppress;   // Program Command to Suppress I/O Fault Alarm
   PCmd_IOFaultUnsuppress : ALIAS FOR IOFault.PCmd_Unsuppress;   // Program Command to Unsuppress I/O Fault Alarm
   PCmd_IOFaultUnshelve : ALIAS FOR IOFault.PCmd_Unshelve;   // Program Command to Unshelve I/O Fault Alarm
   MCmd_Rel : ALIAS FOR CmdSrc.MCmd_Rel;
   OCmd_Unlock : ALIAS FOR CmdSrc.OCmd_Unlock;
   XCmd_On : BOOL;   // External Command to turn device ON
   XCmd_Off : BOOL;   // External Command to turn device OFF
   XCmd_OnPulse : BOOL;   // External Command to pulse device (which is OFF) ON once
   XCmd_OffPulse : BOOL;   // External Command to pulse device (which is ON) OFF once
   XCmd_ContPulse : BOOL;   // External Command to pulse device continuously (blink)
   XCmd_Acq : ALIAS FOR CmdSrc.XCmd_Acq;
   XCmd_Rel : ALIAS FOR CmdSrc.XCmd_Rel;
   XCmd_Reset : BOOL;   // Ext Cmd to clear shed latches and cleared alarms
END_VAR
VAR_OUTPUT
   Out : BOOL; {access Read Only, visible}   // Primary Output 1=ON, 0=OFF
   Out_Horn : BOOL; {access Read Only, visible}   // 1=Sound audible prior to commanded energize/ state change
   SrcQ_IO : DINT; {access Read Only}   // Source and Quality of primary I/O (enumeration)
   SrcQ : DINT; {access Read Only}   // Source and Quality of primary Val/Sts (enumeration)
   Val_Cmd : DINT; {access Read Only}   // Device Command: 0=None, 1=Off, 2=On, 3=Pulse Off, 4=Pulse On, 5=Pulse Cont
   Val_Fdbk : DINT; {access Read Only}   // Device Feedback: 0=Transition, 1=Off, 2=On, 3=Invalid
   Val_Sts : DINT; {access Read Only}   // Device Status 0=off 1=on 2=pulse off 3=pulse on 4=pulse cont. 5=turning off 6=turning on
   Val_Fault : DINT; {access Read Only}   // Device Fault Status 0=none, 16=Feedback Fault, 32=I/O Fault, 34=Config Error
   Val_State : DINT; {access Read Only}   // Internal Logic State (for animating STD on faceplate), see manual
   Val_NotifyAll : DINT; {access Read Only}   // Highest Alarm prio and ack status this object + attached (enum)
   Val_UnackAlmC : DINT; {access Read Only}   // Count of Unacknowledged Alarms
   Val_Owner : DINT; {access Read Only}   // Current Object Owner ID (0=not owned)
   Sts_Out : BOOL; {access Read Only, visible}   // 1=Output is ON (energized), 0=Output is OFF (de-energized)
   Sts_Pulsing : BOOL; {access Read Only, visible}   // 1=Output is in a pusling sequence
   Sts_Horn : BOOL; {access Read Only}   // 1=Horn Active
   Sts_FdbkOff : BOOL; {access Read Only}   // 1=Device Feedback shows device in OFF state
   Sts_FdbkOn : BOOL; {access Read Only}   // 1=Device Feedback shows device in ON state
   Sts_FdbkFail : BOOL; {access Read Only}   // 1=Feedbacks are in an INVALID state (not ON, OFF or TRANSIT)
   Sts_Available : BOOL; {access Read Only}   // 1=Device available for control by automation (Prog)
   Sts_Bypass : BOOL; {access Read Only}   // 1=Bypassable Interlocks and Permissives are Bypassed
   Sts_BypActive : BOOL; {access Read Only}   // 1=Interlock / Permissive Bypassing Active (Bypassed or Maintenance)
   Sts_NotRdy : BOOL; {access Read Only}   // 1=Device Not Ready, see detail bits for reason
   Nrdy_CfgErr : BOOL; {access Read Only}   // 1=Device Not Ready: Configuration Error
   Nrdy_Fail : BOOL; {access Read Only}   // 1=Device Not Ready: Device Failure (Shed Requires Reset)
   Nrdy_Intlk : BOOL; {access Read Only}   // 1=Device Not Ready: Interlock Not OK
   Nrdy_IOFault : BOOL; {access Read Only}   // 1=Device Not Ready: I/O Fault (Shed Requires Reset)
   Nrdy_OoS : BOOL; {access Read Only}   // 1=Device Not Ready: Device is Out of Service
   Nrdy_PrioOff : BOOL; {access Read Only}   // 1=Device Not Ready: Oper/Ext Priority Off Comand Requires Reset
   Nrdy_Perm : BOOL; {access Read Only}   // 1=Device Not Ready: Permissive Not OK
   Sts_MaintByp : BOOL; {access Read Only}   // 1=Device has a Maintenance Bypass function active
   Sts_AlmInh : BOOL; {access Read Only}   // 1=One or more Alarms Shelved, Disabled or Suppressed
   Sts_Err : BOOL; {access Read Only, visible}   // 1=Error in Config: see detail bits for reason
   Err_Timer : BOOL; {access Read Only}   // 1=Error in Config: Feeback Check timer preset (use 0 to 2147483)
   Err_Sim : BOOL; {access Read Only}   // 1=Error in Config: Simulation timer preset (use 0 to 2147483)
   Err_Alarm : BOOL; {access Read Only}   // 1=Error in Config: Alarm Min On Time, Shelf Time, Severity
   Sts_Hand : ALIAS FOR CmdSrc.Sts_Hand; {access Read Only, visible}
   Sts_OoS : ALIAS FOR CmdSrc.Sts_OoS; {access Read Only, visible}
   Sts_Maint : ALIAS FOR CmdSrc.Sts_Maint; {access Read Only, visible}
   Sts_Ovrd : ALIAS FOR CmdSrc.Sts_Ovrd; {access Read Only, visible}
   Sts_Ext : ALIAS FOR CmdSrc.Sts_Ext; {access Read Only, visible}
   Sts_Prog : ALIAS FOR CmdSrc.Sts_Prog; {access Read Only, visible}
   Sts_ProgLocked : ALIAS FOR CmdSrc.Sts_ProgLocked; {access Read Only}
   Sts_Oper : ALIAS FOR CmdSrc.Sts_Oper; {access Read Only, visible}
   Sts_OperLocked : ALIAS FOR CmdSrc.Sts_OperLocked; {access Read Only}
   Sts_Normal : ALIAS FOR CmdSrc.Sts_Normal; {access Read Only}
   Sts_ExtReqInh : ALIAS FOR CmdSrc.Sts_ExtReqInh; {access Read Only}
   Sts_ProgReqInh : ALIAS FOR CmdSrc.Sts_ProgReqInh; {access Read Only}
   Sts_MAcqRcvd : ALIAS FOR CmdSrc.Sts_MAcqRcvd; {access Read Only}
   Sts_RdyReset : ALIAS FOR ORdy_Reset; {access Read Only}   // 1=A latched alarm or shed condition is ready to be reset
   Sts_RdyAck : BOOL; {access Read Only}   // 1=An alarm is ready to be acknowledged
   Sts_OnFail : ALIAS FOR OnFail.Inp;   // 1=Device Failed to Turn ON
   Alm_OnFail : ALIAS FOR OnFail.Alm;   // 1=Device Fail to Turn ON Alarm
   Ack_OnFail : ALIAS FOR OnFail.Ack;   // 1=Fail to Turn ON Alarm has been acknowledged
   Sts_OnFailDisabled : ALIAS FOR OnFail.Disabled;   // 1=Fail to Turn ON Alarm has been Disabled by Maintenance
   Sts_OnFailShelved : ALIAS FOR OnFail.Shelved;   // 1=Fail to Turn ON Alarm has been Shelved by Operator
   Sts_OnFailSuppressed : ALIAS FOR OnFail.Suppressed;   // 1=Fail to Turn ON Alarm has been Suppressed by Program
   Sts_OffFail : ALIAS FOR OffFail.Inp;   // 1=Device Failed to Turn OFF
   Alm_OffFail : ALIAS FOR OffFail.Alm;   // 1=Device Fail to Turn OFF Alarm
   Ack_OffFail : ALIAS FOR OffFail.Ack;   // 1=Fail to Turn OFF Alarm has been acknowledged
   Sts_OffFailDisabled : ALIAS FOR OffFail.Disabled;   // 1=Fail to Turn OFF Alarm has been Disabled by Maintenance
   Sts_OffFailShelved : ALIAS FOR OffFail.Shelved;   // 1=Fail to Turn OFF Alarm has been Shelved by Operator
   Sts_OffFailSuppressed : ALIAS FOR OffFail.Suppressed;   // 1=Fail to Turn OFF Alarm has been Suppressed by Program
   Sts_IntlkTrip : ALIAS FOR IntlkTrip.Inp;   // 1=Device turned OFF by an Interlock NOT OK (one-shot)
   Alm_IntlkTrip : ALIAS FOR IntlkTrip.Alm;   // 1=Alarm: Device turned OFF by an Interlock NOT OK
   Ack_IntlkTrip : ALIAS FOR IntlkTrip.Ack;   // 1=Interlock Trip Alarm has been acknowledged
   Sts_IntlkTripDisabled : ALIAS FOR IntlkTrip.Disabled;   // 1=Interlock Trip Alarm has been Disabled by Maintenance
   Sts_IntlkTripShelved : ALIAS FOR IntlkTrip.Shelved;   // 1=Interlock Trip Alarm has been Shelved by Operator
   Sts_IntlkTripSuppressed : ALIAS FOR IntlkTrip.Suppressed;   // 1=Interlock Trip Alarm has been Suppressed by Program
   Sts_IOFault : ALIAS FOR IOFault.Inp;   // I/O Comm Fault Status (0=OK, 1=Bad)
   Alm_IOFault : ALIAS FOR IOFault.Alm;   // 1=I/O Fault Alarm
   Ack_IOFault : ALIAS FOR IOFault.Ack;   // 1=I/O Fault Alarm has been acknowledged
   Sts_IOFaultDisabled : ALIAS FOR IOFault.Disabled;   // 1=I/O Fault Alarm has been Disabled by Maintenance
   Sts_IOFaultShelved : ALIAS FOR IOFault.Shelved;   // 1=I/O Fault Alarm has been Shelved by Operator
   Sts_IOFaultSuppressed : ALIAS FOR IOFault.Suppressed;   // 1=I/O Fault Alarm has been Suppressed by Program
   MRdy_Rel : ALIAS FOR CmdSrc.MRdy_Rel; {access Read Only}
   ORdy_Unlock : ALIAS FOR CmdSrc.ORdy_Unlock; {access Read Only}
   P_DOut : BOOL;   // Unique Parameter Name for auto - discovery
END_VAR
VAR
   Wrk_OffT : TIMER; {access Read Only}   // Off Feedback Check Timer
   Wrk_OnT : TIMER; {access Read Only}   // On Feedback Check Timer
   Wrk_SimOffT : TIMER; {access None}   // Simulation Delay until OFF
   Wrk_SimOnT : TIMER; {access None}   // Simulation Delay until ON
   Wrk_OnFdbk : BOOL; {access None}   // ON Feedback based on Command Source, simulation, etc. 1=confirmed ON
   Wrk_Notify : DINT; {access None}   // Buffer for building Val_Notify
   Wrk_Bypass : BOOL; {access None}   // Internal Bypassable Permissives and Interlocks are Bypassed flag
   CmdSrc : P_CmdSrc := (Cfg_HasOper := 1, Cfg_HasOperLocked := 1, Cfg_HasProg := 1, Cfg_HasProgLocked := 1, Cfg_HasMaint := 1, Cfg_HasMOoS := 1, Cfg_OvrdOverLock := 1, Sts_Oper := 1);   // Control / Command Source Selection
   IOFault : P_Alarm := (Cfg_AckReqd := 1, Cfg_AllowShelve := 1, Cfg_AllowDisable := 1, Cfg_Severity := 1000, Cfg_AlmMinOnT := 5, PCfg_AllowExist := 1, Ack := 1);   // I/O Fault Alarm
   IntlkTrip : P_Alarm := (Cfg_AckReqd := 1, Cfg_AllowShelve := 1, Cfg_AllowDisable := 1, Cfg_Severity := 500, Cfg_AlmMinOnT := 5, PCfg_AllowExist := 1, Ack := 1);   // Interlock Trip Alarm
   OffFail : P_Alarm := (Cfg_AckReqd := 1, Cfg_AllowShelve := 1, Cfg_AllowDisable := 1, Cfg_Severity := 1000, Cfg_AlmMinOnT := 5, PCfg_AllowExist := 1, Ack := 1);   // Device Failed to Turn OFF Alarm
   OnFail : P_Alarm := (Cfg_AckReqd := 1, Cfg_AllowShelve := 1, Cfg_AllowDisable := 1, Cfg_Severity := 1000, Cfg_AlmMinOnT := 5, PCfg_AllowExist := 1, Ack := 1);   // Device Failed to Turn ON Alarm
   Cfg_Tag : STRING_20 := 'P_DOut';   // Tagname for display on HMI
   Cfg_Label : STRING_20 := 'Discrete Device';   // Label for graphic symbol displayed on HMI
   Cfg_Desc : STRING_40 := 'Discrete On/Off Device';   // Description for display on HMI
   Wrk_OffFdbk : BOOL; {access None}   // OFF Feedback based on Command Source, simulation, etc. 1=confirmed OFF
   Wrk_OnPulseT : TIMER; {access Read Only}   // Output ON Pulse Timer
   Wrk_OffPulseT : TIMER; {access Read Only}   // Output OFF Pulse Timer
   Wrk_OffDelayT : TIMER; {access Read Only}   // Dealy before turning output OFF (Timer)
   Wrk_OnDelayT : TIMER; {access Read Only}   // Delay before turning output ON (Timer)
   Wrk_PermOK : BOOL; {access None}   // 1=Permissives are all OK to energize
   HMI_Tab : SINT;   // Tab to display (FTView ME)
   Wrk_Cmd : DINT; {access None}   // Device Command: 0= None, bit .0=Off, bit .1=On, bit .2=Pulse Off, bit .3=Pulse On, bit .4=Pulse Cont.
   Wrk_Fault : DINT; {access None}   // Buffer for building Val_Fault
   Wrk_SrcQ : DINT; {access None}   // Register for building Source / Quality enumeration
   Cfg_1StText : STRING_8 := 'On';   // Text to display in PV=1 State
   Cfg_0StText : STRING_8 := 'Off';   // Text to display in PV=0 State
   HMI_Type : STRING_16 := 'P_DOut'; {access Read Only}   // Type identifier for HMI navigation
   HMI_Lib : STRING_12 := 'RA-BAS'; {access Read Only}   // Display Library for Faceplate call-up
   Wrk_NotRdy : BOOL; {access None}   // Device Not Ready conditions excluding shed latches
   Wrk_NoLongerSim : BOOL; {access None}   // Switched from Simulated to Real Device this scan
   Cfg_Area : STRING_Area := 'area01';   // Process Area for security
   Wrk_UnackAlmC : DINT; {access None}   // Buffer for building Val_UnackAlmC
   Val_Notify : DINT; {access Read Only}   // Current Alarm Level and Acknowledgement (enumeration)
   OCmd_ResetAckAll : BOOL;   // Operator Command to Reset all Alarms and latched Shed conditions
   OCmd_Reset : BOOL;   // Operator Command to Reset all Alarms requiring Reset
   OCmd_ContPulse : BOOL;   // Operator Command to pulse device continuously (blink)
   OCmd_OffPulse : BOOL;   // Operator Command to pulse device (which is ON) OFF once
   OCmd_OnPulse : BOOL;   // Operator Command to pulse device (which is OFF) ON once
   OCmd_Off : BOOL;   // Operator Command to turn device OFF
   OCmd_On : BOOL;   // Operator Command to turn device ON
   MCmd_Check : BOOL;   // Maintenance Command to Check (not bypass) all Interlocks and Permissives
   MCmd_Bypass : BOOL;   // Maintenance Command to Bypass all Bypassable Interlocks and Permissives
   ORdy_ResetAckAll : BOOL; {access Read Only}   // 1=Ready for OCmd_ResetAckAll (enables HMI button)
   ORdy_Reset : BOOL; {access Read Only}   // 1=Ready for OCmd_Reset (enables HMI button)
   ORdy_ContPulse : BOOL; {access Read Only}   // 1=Ready for OCmd_ContPulse (enables HMI button)
   ORdy_OffPulse : BOOL; {access Read Only}   // 1=Ready for OCmd_OffPulse (enables HMI button)
   ORdy_OnPulse : BOOL; {access Read Only}   // 1=Ready for OCmd_OnPulse (enables HMI button)
   ORdy_Off : BOOL; {access Read Only}   // 1=Ready for OCmd_Off (enables HMI button)
   ORdy_On : BOOL; {access Read Only}   // 1=Ready for OCmd_On (enables HMI button)
   MRdy_Check : BOOL; {access Read Only}   // 1=Ready for MCmd_Check (enables HMI button)
   MRdy_Bypass : BOOL; {access Read Only}   // 1=Ready for MCmd_Bypass (enables HMI button)
   Wrk_State : DINT; {access None}   // Internal value of state machine current state
   Wrk_StartHornT : TIMER; {access None}   // Timer for audible alert or start
   Wrk_StartHorn : BOOL; {access None}   // 1=Sound audible prior to commanded energize/ state change
END_VAR

ROUTINE EnableInFalse   (* ladder *)
// Out of Service; output is OFF; feedback Status shown if available; Alarms inhibited.
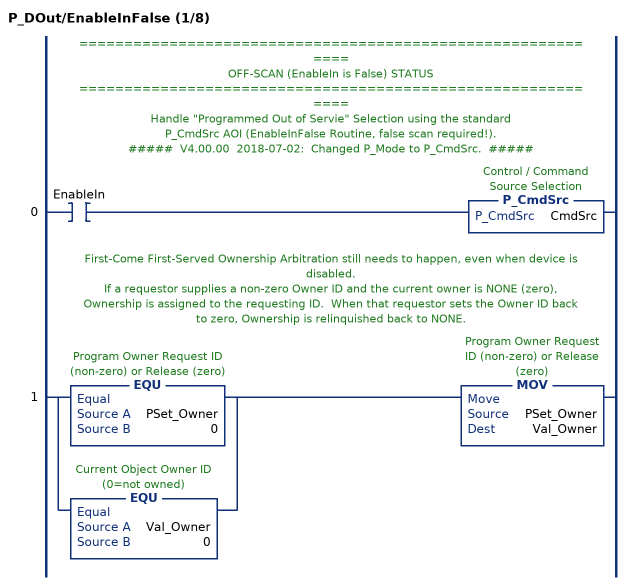
   // ============================================================
   // OFF-SCAN (EnableIn is False) STATUS
   // ============================================================
   // Handle "Programmed Out of Servie" Selection using the standard
   // P_CmdSrc AOI (EnableInFalse Routine, false scan required!).
   // #####  V4.00.00  2018-07-02:  Changed P_Mode to P_CmdSrc.  #####
   0: XIC(EnableIn)P_CmdSrc(CmdSrc);
   // First-Come First-Served Ownership Arbitration still needs to happen, even when device is disabled.
   // If a requestor supplies a non-zero Owner ID and the current owner is NONE (zero),
   // Ownership is assigned to the requesting ID.  When that requestor sets the Owner ID back
   // to zero, Ownership is relinquished back to NONE.
   1: [EQU(PSet_Owner,0) ,EQU(Val_Owner,0) ]MOV(PSet_Owner,Val_Owner);
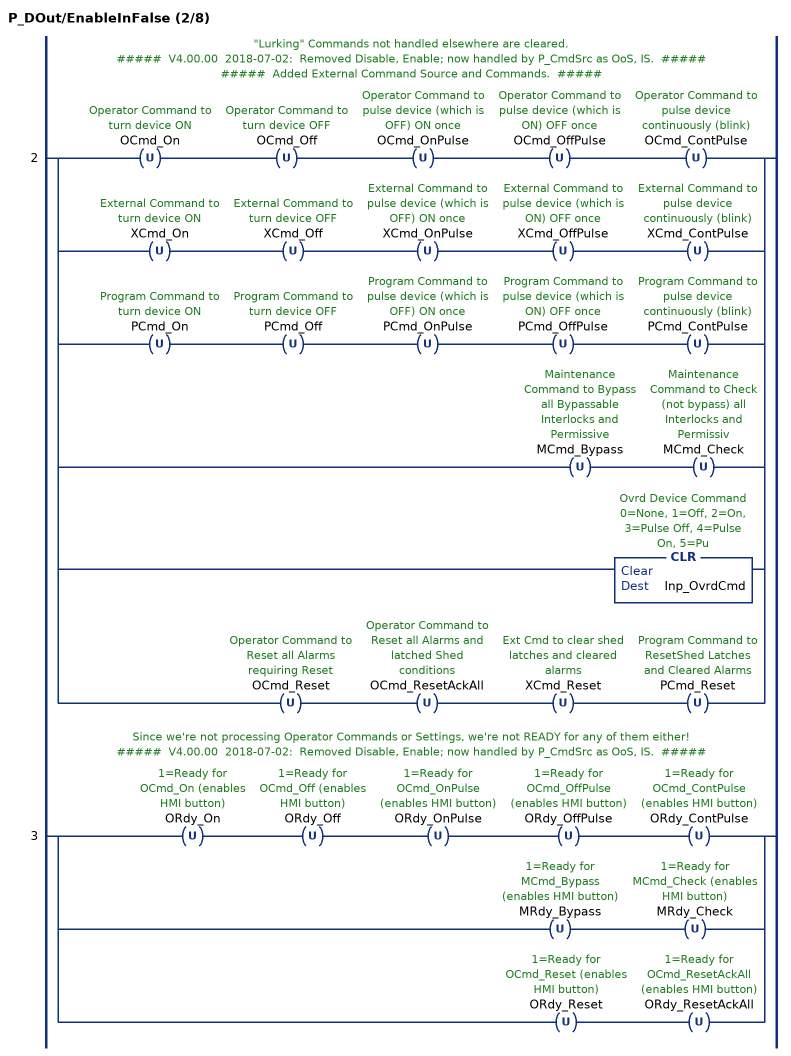
   // "Lurking" Commands not handled elsewhere are cleared.
   // #####  V4.00.00  2018-07-02:  Removed Disable, Enable; now handled by P_CmdSrc as OoS, IS.  #####
   // #####  Added External Command Source and Commands.  #####
   2: [OTU(OCmd_On) OTU(OCmd_Off) OTU(OCmd_OnPulse) OTU(OCmd_OffPulse) OTU(OCmd_ContPulse) ,OTU(XCmd_On) OTU(XCmd_Off) OTU(XCmd_OnPulse) OTU(XCmd_OffPulse) OTU(XCmd_ContPulse) ,OTU(PCmd_On) OTU(PCmd_Off) OTU(PCmd_OnPulse) OTU(PCmd_OffPulse) OTU(PCmd_ContPulse) ,OTU(MCmd_Bypass) OTU(MCmd_Check) ,CLR(Inp_OvrdCmd) ,OTU(OCmd_Reset) OTU(OCmd_ResetAckAll) OTU(XCmd_Reset) OTU(PCmd_Reset) ];
   // Since we're not processing Operator Commands or Settings, we're not READY for any of them either!
   // #####  V4.00.00  2018-07-02:  Removed Disable, Enable; now handled by P_CmdSrc as OoS, IS.  #####
   3: [OTU(ORdy_On) OTU(ORdy_Off) OTU(ORdy_OnPulse) OTU(ORdy_OffPulse) OTU(ORdy_ContPulse) ,OTU(MRdy_Bypass) OTU(MRdy_Check) ,OTU(ORdy_Reset) OTU(ORdy_ResetAckAll) ];
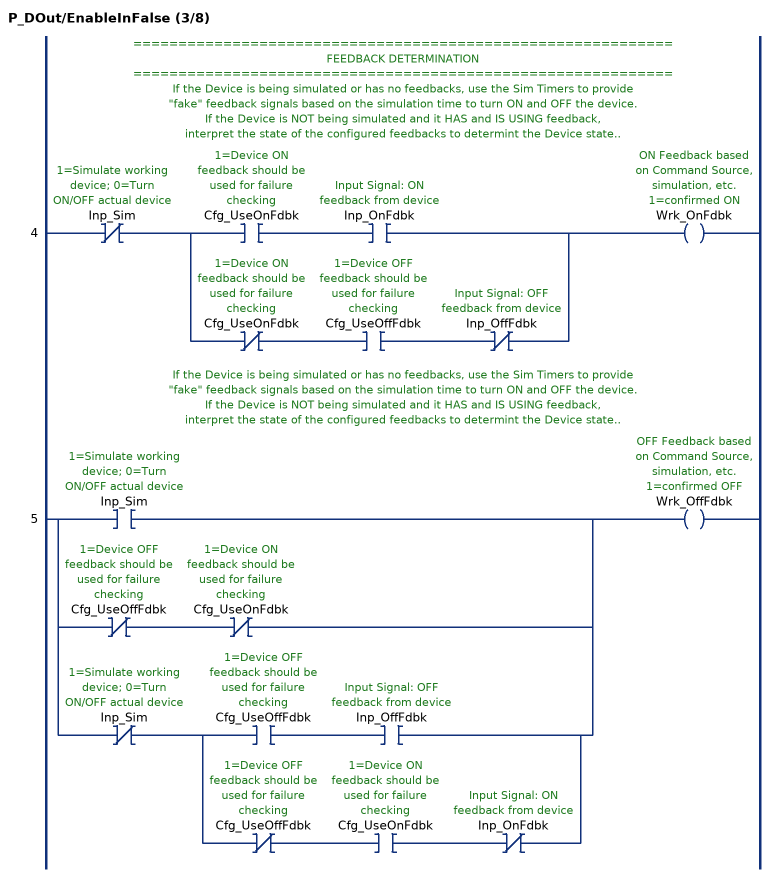
   // ============================================================
   // FEEDBACK DETERMINATION
   // ============================================================
   // If the Device is being simulated or has no feedbacks, use the Sim Timers to provide
   // "fake" feedback signals based on the simulation time to turn ON and OFF the device.
   // If the Device is NOT being simulated and it HAS and IS USING feedback,
   // interpret the state of the configured feedbacks to determint the Device state..
   4: XIO(Inp_Sim)[XIC(Cfg_UseOnFdbk) XIC(Inp_OnFdbk) ,XIO(Cfg_UseOnFdbk) XIC(Cfg_UseOffFdbk) XIO(Inp_OffFdbk) ]OTE(Wrk_OnFdbk);
   // If the Device is being simulated or has no feedbacks, use the Sim Timers to provide
   // "fake" feedback signals based on the simulation time to turn ON and OFF the device.
   // If the Device is NOT being simulated and it HAS and IS USING feedback,
   // interpret the state of the configured feedbacks to determint the Device state..
   5: [[XIC(Inp_Sim) ,XIO(Cfg_UseOffFdbk) XIO(Cfg_UseOnFdbk) ] ,XIO(Inp_Sim) [XIC(Cfg_UseOffFdbk) XIC(Inp_OffFdbk) ,XIO(Cfg_UseOffFdbk) XIC(Cfg_UseOnFdbk) XIO(Inp_OnFdbk) ] ]OTE(Wrk_OffFdbk);
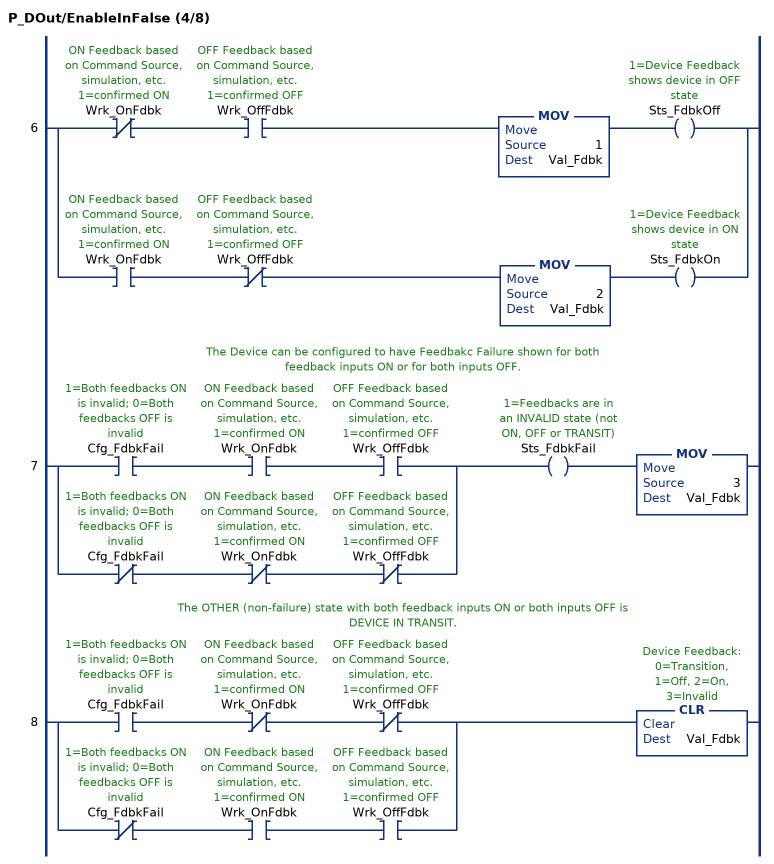
   6: [XIO(Wrk_OnFdbk) XIC(Wrk_OffFdbk) MOV(1,Val_Fdbk) OTE(Sts_FdbkOff) ,XIC(Wrk_OnFdbk) XIO(Wrk_OffFdbk) MOV(2,Val_Fdbk) OTE(Sts_FdbkOn) ];
   // The Device can be configured to have Feedbakc Failure shown for both
   // feedback inputs ON or for both inputs OFF.
   7: [XIC(Cfg_FdbkFail) XIC(Wrk_OnFdbk) XIC(Wrk_OffFdbk) ,XIO(Cfg_FdbkFail) XIO(Wrk_OnFdbk) XIO(Wrk_OffFdbk) ]OTE(Sts_FdbkFail)MOV(3,Val_Fdbk);
   // The OTHER (non-failure) state with both feedback inputs ON or both inputs OFF is
   // DEVICE IN TRANSIT.
   8: [XIC(Cfg_FdbkFail) XIO(Wrk_OnFdbk) XIO(Wrk_OffFdbk) ,XIO(Cfg_FdbkFail) XIC(Wrk_OnFdbk) XIC(Wrk_OffFdbk) ]CLR(Val_Fdbk);
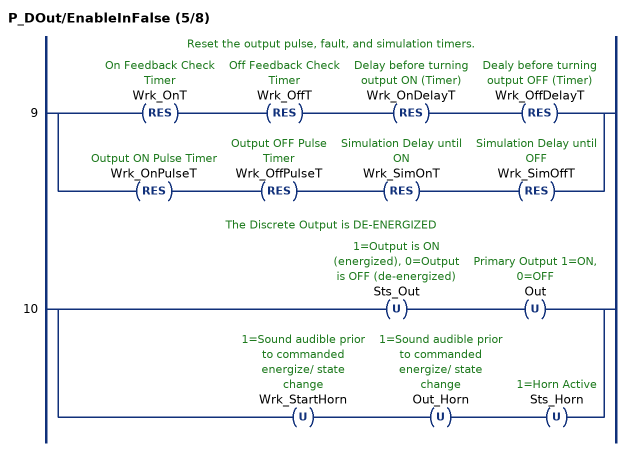
   // Reset the output pulse, fault, and simulation timers.
   9: [RES(Wrk_OnT) RES(Wrk_OffT) RES(Wrk_OnDelayT) RES(Wrk_OffDelayT) ,RES(Wrk_OnPulseT) RES(Wrk_OffPulseT) RES(Wrk_SimOnT) RES(Wrk_SimOffT) ];
   // The Discrete Output is DE-ENERGIZED
   10: [OTU(Sts_Out) OTU(Out) ,OTU(Wrk_StartHorn) OTU(Out_Horn) OTU(Sts_Horn) ];
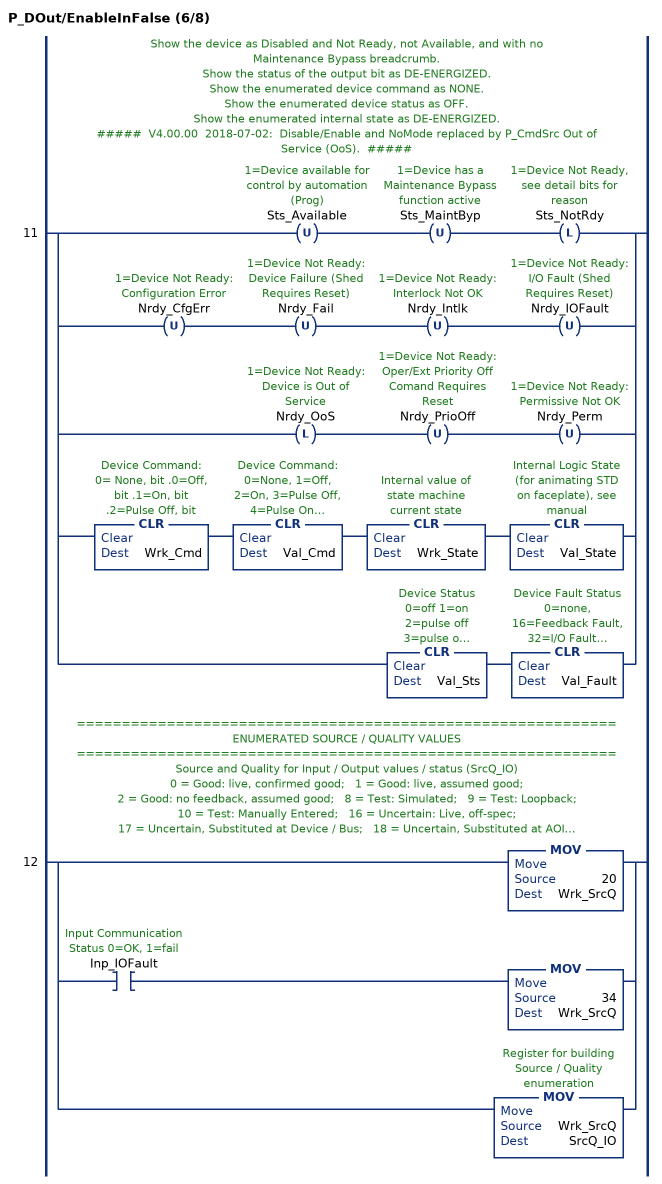
   // Show the device as Disabled and Not Ready, not Available, and with no
   // Maintenance Bypass breadcrumb.
   // Show the status of the output bit as DE-ENERGIZED.
   // Show the enumerated device command as NONE.
   // Show the enumerated device status as OFF.
   // Show the enumerated internal state as DE-ENERGIZED.
   // #####  V4.00.00  2018-07-02:  Disable/Enable and NoMode replaced by P_CmdSrc Out of Service (OoS).  #####
   11: [OTU(Sts_Available) OTU(Sts_MaintByp) OTL(Sts_NotRdy) ,OTU(Nrdy_CfgErr) OTU(Nrdy_Fail) OTU(Nrdy_Intlk) OTU(Nrdy_IOFault) ,OTL(Nrdy_OoS) OTU(Nrdy_PrioOff) OTU(Nrdy_Perm) ,CLR(Wrk_Cmd) CLR(Val_Cmd) CLR(Wrk_State) CLR(Val_State) ,CLR(Val_Sts) CLR(Val_Fault) ];
   // ============================================================
   // ENUMERATED SOURCE / QUALITY VALUES
   // ============================================================
   // Source and Quality for Input / Output values / status (SrcQ_IO)
   // 0 = Good: live, confirmed good;   1 = Good: live, assumed good;
   // 2 = Good: no feedback, assumed good;   8 = Test: Simulated;   9 = Test: Loopback;
   // 10 = Test: Manually Entered;   16 = Uncertain: Live, off-spec;
   // 17 = Uncertain, Substituted at Device / Bus;   18 = Uncertain, Substituted at AOI;
   // 19 = Uncertain, using last known good;    20 = Uncertain, using replacement value;
   // 32 = Bad, Signal Failure;   33 = Bad, Channel Fault;
   // 34 = Bad, Module / Comms Fault;   35 = Bad, Invalid Configuration
   12: [MOV(20,Wrk_SrcQ) ,XIC(Inp_IOFault) MOV(34,Wrk_SrcQ) ,MOV(Wrk_SrcQ,SrcQ_IO) ];
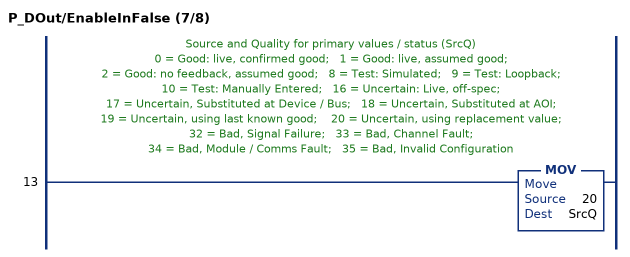
   // Source and Quality for primary values / status (SrcQ)
   // 0 = Good: live, confirmed good;   1 = Good: live, assumed good;
   // 2 = Good: no feedback, assumed good;   8 = Test: Simulated;   9 = Test: Loopback;
   // 10 = Test: Manually Entered;   16 = Uncertain: Live, off-spec;
   // 17 = Uncertain, Substituted at Device / Bus;   18 = Uncertain, Substituted at AOI;
   // 19 = Uncertain, using last known good;    20 = Uncertain, using replacement value;
   // 32 = Bad, Signal Failure;   33 = Bad, Channel Fault;
   // 34 = Bad, Module / Comms Fault;   35 = Bad, Invalid Configuration
   13: MOV(20,SrcQ);
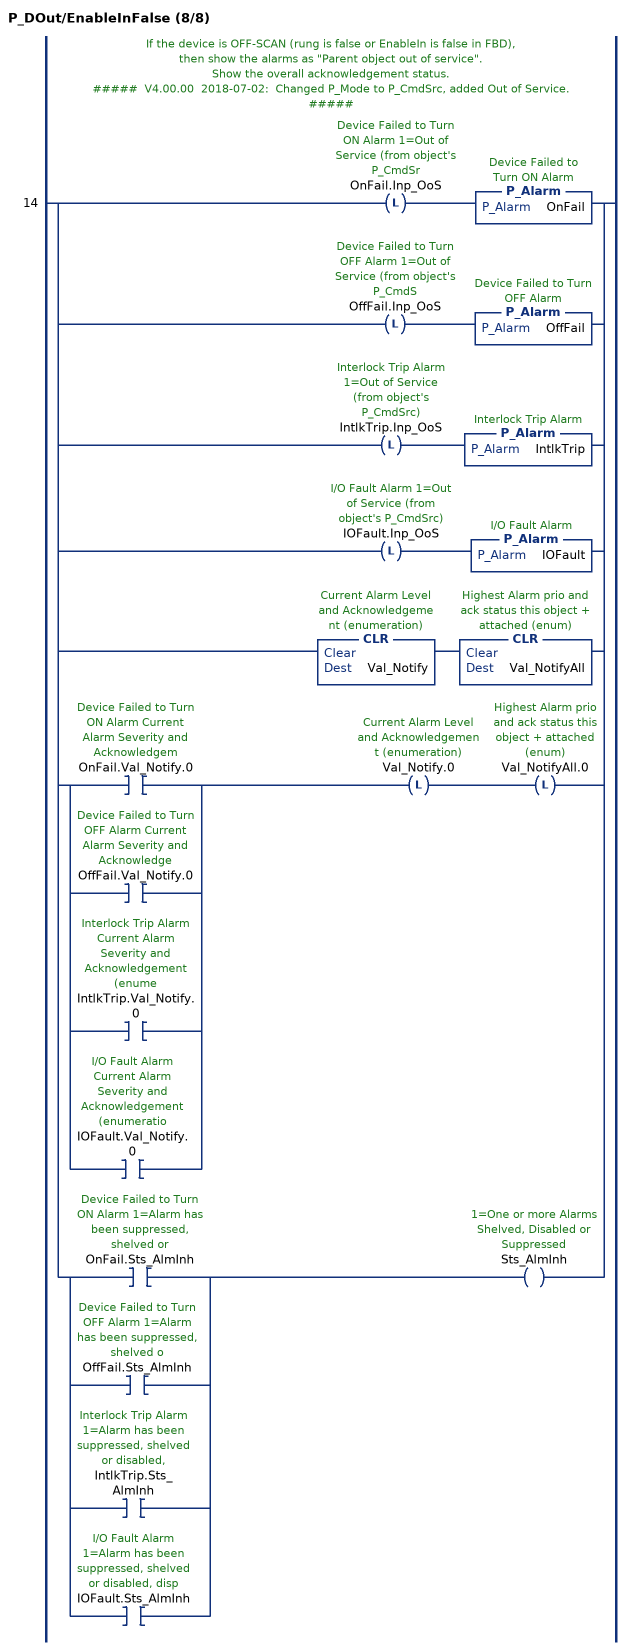
   // If the device is OFF-SCAN (rung is false or EnableIn is false in FBD),
   // then show the alarms as "Parent object out of service".
   // Show the overall acknowledgement status.
   // #####  V4.00.00  2018-07-02:  Changed P_Mode to P_CmdSrc, added Out of Service.  #####
   14: [OTL(OnFail.Inp_OoS) P_Alarm(OnFail) ,OTL(OffFail.Inp_OoS) P_Alarm(OffFail) ,OTL(IntlkTrip.Inp_OoS) P_Alarm(IntlkTrip) ,OTL(IOFault.Inp_OoS) P_Alarm(IOFault) ,CLR(Val_Notify) CLR(Val_NotifyAll) ,[XIC(OnFail.Val_Notify.0) ,XIC(OffFail.Val_Notify.0) ,XIC(IntlkTrip.Val_Notify.0) ,XIC(IOFault.Val_Notify.0) ] OTL(Val_Notify.0) OTL(Val_NotifyAll.0) ,[XIC(OnFail.Sts_AlmInh) ,XIC(OffFail.Sts_AlmInh) ,XIC(IntlkTrip.Sts_AlmInh) ,XIC(IOFault.Sts_AlmInh) ] OTE(Sts_AlmInh) ];
END_ROUTINE
